// ---- DUTs/UR_6_T2O_IntRegisters/UR_6_T2O_IntRegisters.TcDUT
TYPE UR_6_T2O_IntRegisters :
STRUCT
INT0:ARRAY[0..3] OF BYTE;
INT1:ARRAY[0..3] OF BYTE;
INT2:ARRAY[0..3] OF BYTE;
INT3:ARRAY[0..3] OF BYTE;
INT4:ARRAY[0..3] OF BYTE;
INT5:ARRAY[0..3] OF BYTE;
INT6:ARRAY[0..3] OF BYTE;
INT7:ARRAY[0..3] OF BYTE;
INT8:ARRAY[0..3] OF BYTE;
INT9:ARRAY[0..3] OF BYTE;
INT10:ARRAY[0..3] OF BYTE;
INT11:ARRAY[0..3] OF BYTE;
INT12:ARRAY[0..3] OF BYTE;
INT13:ARRAY[0..3] OF BYTE;
INT14:ARRAY[0..3] OF BYTE;
INT15:ARRAY[0..3] OF BYTE;
INT16:ARRAY[0..3] OF BYTE;
INT17:ARRAY[0..3] OF BYTE;
INT18:ARRAY[0..3] OF BYTE;
INT19:ARRAY[0..3] OF BYTE;
INT20:ARRAY[0..3] OF BYTE;
INT21:ARRAY[0..3] OF BYTE;
INT22:ARRAY[0..3] OF BYTE;
INT23:ARRAY[0..3] OF BYTE;
END_STRUCT
END_TYPE

// ---- DUTs/UR_7_T2O_FloatRegisters/UR_7_T2O_FloatRegisters.TcDUT
TYPE UR_7_T2O_FloatRegisters :
	
STRUCT
FLOAT0:ARRAY[0..3] OF BYTE;
FLOAT1:ARRAY[0..3] OF BYTE;
FLOAT2:ARRAY[0..3] OF BYTE;
FLOAT3:ARRAY[0..3] OF BYTE;
FLOAT4:ARRAY[0..3] OF BYTE;
FLOAT5:ARRAY[0..3] OF BYTE;
FLOAT6:ARRAY[0..3] OF BYTE;
FLOAT7:ARRAY[0..3] OF BYTE;
FLOAT8:ARRAY[0..3] OF BYTE;
FLOAT9:ARRAY[0..3] OF BYTE;
FLOAT10:ARRAY[0..3] OF BYTE;
FLOAT11:ARRAY[0..3] OF BYTE;
FLOAT12:ARRAY[0..3] OF BYTE;
FLOAT13:ARRAY[0..3] OF BYTE;
FLOAT14:ARRAY[0..3] OF BYTE;
FLOAT15:ARRAY[0..3] OF BYTE;
FLOAT16:ARRAY[0..3] OF BYTE;
FLOAT17:ARRAY[0..3] OF BYTE;
FLOAT18:ARRAY[0..3] OF BYTE;
FLOAT19:ARRAY[0..3] OF BYTE;
FLOAT20:ARRAY[0..3] OF BYTE;
FLOAT21:ARRAY[0..3] OF BYTE;
FLOAT22:ARRAY[0..3] OF BYTE;
FLOAT23:ARRAY[0..3] OF BYTE;
END_STRUCT
END_TYPE

// ---- DUTs/UR_9_O2T_Registers/UR_9_O2T_Registers.TcDUT
TYPE UR_9_O2T_Registers :
STRUCT
	  Bits : UR_O2T_bits;
      Ints : UR_O2T_int;
      Floats : UR_O2T_floats;
END_STRUCT
END_TYPE

// ---- DUTs/UR_9_O2T_Registers/UR_O2T_bits.TcDUT
TYPE UR_O2T_bits :
   STRUCT
	B0:BIT;
	B1:BIT;
	B2:BIT;
	B3:BIT;
	B4:BIT;
	B5:BIT;
	B6:BIT;
	B7:BIT;
	B8:BIT;
	B9:BIT;
	B10:BIT;
	B11:BIT;
	B12:BIT;
	B13:BIT;
	B14:BIT;
	B15:BIT;
	B16:BIT;
	B17:BIT;
	B18:BIT;
	B19:BIT;
	B20:BIT;
	B21:BIT;
	B22:BIT;
	B23:BIT;
	B24:BIT;
	B25:BIT;
	B26:BIT;
	B27:BIT;
	B28:BIT;
	B29:BIT;
	B30:BIT;
	B31:BIT;
   END_STRUCT
END_TYPE

// ---- DUTs/UR_9_O2T_Registers/UR_O2T_floats.TcDUT
TYPE UR_O2T_floats :
STRUCT
FLOAT0:ARRAY[0..3] OF BYTE;
FLOAT1:ARRAY[0..3] OF BYTE;
FLOAT2:ARRAY[0..3] OF BYTE;
FLOAT3:ARRAY[0..3] OF BYTE;
FLOAT4:ARRAY[0..3] OF BYTE;
FLOAT5:ARRAY[0..3] OF BYTE;
FLOAT6:ARRAY[0..3] OF BYTE;
FLOAT7:ARRAY[0..3] OF BYTE;
FLOAT8:ARRAY[0..3] OF BYTE;
FLOAT9:ARRAY[0..3] OF BYTE;
FLOAT10:ARRAY[0..3] OF BYTE;
FLOAT11:ARRAY[0..3] OF BYTE;
END_STRUCT
END_TYPE

// ---- DUTs/UR_9_O2T_Registers/UR_O2T_int.TcDUT
TYPE UR_O2T_int :
STRUCT
INT0:ARRAY[0..3] OF BYTE;
INT1:ARRAY[0..3] OF BYTE;
INT2:ARRAY[0..3] OF BYTE;
INT3:ARRAY[0..3] OF BYTE;
INT4:ARRAY[0..3] OF BYTE;
INT5:ARRAY[0..3] OF BYTE;
INT6:ARRAY[0..3] OF BYTE;
INT7:ARRAY[0..3] OF BYTE;
INT8:ARRAY[0..3] OF BYTE;
INT9:ARRAY[0..3] OF BYTE;
INT10:ARRAY[0..3] OF BYTE;
INT11:ARRAY[0..3] OF BYTE;
END_STRUCT
END_TYPE

// ---- DUTs/Vision Struct/ck_real_flag_data.TcDUT
//struct to return values from POUS->Vision_functions->wr_real_value f
TYPE ck_real_flag_data :
STRUCT
	Flag : BOOL;
	Value : REAL;
END_STRUCT
END_TYPE

// ---- DUTs/Vision Struct/Vision_data.TcDUT
//struct to save vision real values system
TYPE Vision_data :
STRUCT
Val1 : REAL:= -1;
Val2 : REAL:= -1;
Val3 : REAL:= -1;
END_STRUCT
END_TYPE

// ---- DUTs/Vision Struct/Vision_flags.TcDUT
//struct to save vision flags values system
TYPE Vision_flags :
STRUCT
Flag1 :BOOL:=FALSE;	
Flag2 :BOOL:=FALSE;	
Flag3 :BOOL:=FALSE;	
END_STRUCT
END_TYPE

// ---- DUTs/Vision Struct/Vision_int_state.TcDUT
TYPE Vision_int_state :
STRUCT
	Val1 : INT:= -1;
	Val2 : INT:= -1;
	Val3 : INT:= -1;
END_STRUCT
END_TYPE

// ---- GVLs/MainProg Params/Constans/VFUNCTION.TcGVL
{attribute 'qualified_only'}
VAR_GLOBAL CONSTANT
	 	
	TEST:INT := 1; //test state one by one
	NORM:INT := 2; // normal functionality
	MOVEMENTS:INT := 3; // test just movements
	CK_COMUNICATIONS:INT := 4; // test all comunication
	POWEROFF:INT := 5; // prepare to poweroff the system
END_VAR

// ---- GVLs/MainProg Params/Constans/_FUNCTION.TcGVL
{attribute 'qualified_only'}
VAR_GLOBAL CONSTANT
	 	
	TEST:INT := 1; //test state one by one
	NORM:INT := 2; // normal functionality
	MOVEMENTS:INT := 3; // test just movements
	CK_COMUNICATIONS:INT := 4; // test all comunication
	POWEROFF:INT := 5; // prepare to poweroff the system
END_VAR

// ---- GVLs/MainProg Params/Variables/GLV_USER_FUN.TcGVL
{attribute 'qualified_only'}
VAR_GLOBAL RETAIN
		Value :INT:=2;
END_VAR

// ---- GVLs/miscellaneus/data_to_robot.TcGVL
{attribute 'qualified_only'}
VAR_GLOBAL
	head_roll_right : REAL;
	head_roll_left : REAL;
	
	
END_VAR

// ---- GVLs/miscellaneus/Global_actual_velocity.TcGVL
{attribute 'qualified_only'}
VAR_GLOBAL
	actual_velocity AT%I*: DINT;

	
	
	
END_VAR

// ---- GVLs/QRob/QrCts.TcGVL
{attribute 'qualified_only'}
VAR_GLOBAL CONSTANT
	MOVESTATE_INIT :INT:= 1;
	
	MOVESTATE_ENABLE :INT:= 2;
	MOVESTATE_ENABLE_F :INT:= 21;
	
	MOVESTATE_ERROR :INT:=3;
	MOVESTATE_ERROR_F :INT:=31;
	
	MOVESTATE_RESET : INT:=4;
	MOVESTATE_RESET_F : INT:=41;
	
	MOVESTATE_MOVABS : INT:=5;
	MOVESTATE_MOVABS_I :INT:=50;
	MOVESTATE_MOVABS_F :INT:=51;
	
	MOVESTATE_HOME:  INT:=6;
	MOVESTATE_HOME_I:  INT:=60;
	MOVESTATE_HOME_F:  INT:=61;
	
	MOVESTATE_CTR_W : INT := 7;
	MOVESTATE_CTR_W_I : INT := 70;
	MOVESTATE_CTR_W_F : INT := 71;
	
	MOVESTATE_TORQUE : INT := 8;
	MOVESTATE_TORQUE_I : INT := 80;
	MOVESTATE_TORQUE_F : INT := 81;
	
	
	MOVESTATE_RELIEF : INT := 9;
	MOVESTATE_RELIEF_I : INT := 90;
	MOVESTATE_RELIEF_F : INT := 91;
	
	OFFSETHOME : INT := 15;
	OFFSETHOME_I : INT := 150;
	OFFSETHOME_F : INT := 151;
	
END_VAR

// ---- GVLs/QRob/Variables/Global_Servo.TcGVL
{attribute 'qualified_only'}
VAR_GLOBAL
	Axis1 : AXIS_REF;
	
END_VAR

// ---- GVLs/QRob/Variables/QrRetVarState.TcGVL
{attribute 'qualified_only'}
VAR_GLOBAL RETAIN
	Actual_GLV_State :INT:=-1;
	Actual_In_State: INT:=-1;
	Actual_POs :REAL:=0;
END_VAR

// ---- GVLs/Robot Params/Constans/RCts.TcGVL
{attribute 'qualified_only'}
VAR_GLOBAL CONSTANT


// 


   

//############### CS.UR3 CONSTANTS STATES ###################
//########################################################
	RESET_STATE:INT:=-1;
	//CS.UR3 states
	UR3:INT:=3;
	UR3Home:INT := 30;
	UR3Home_I :INT:= 300;
	UR3Home_F :INT:= 301;
	
    UR3CatchSeparator:INT := 31;
	UR3CatchSeparator_I:INT := 310;
	UR3CatchSeparator_F:INT := 311;
	
	UR3Move:INT := 32;
	UR3Move_I:INT := 320;	
	UR3Move_F:INT := 321;
	
	UR3DropBench:INT := 33;
	UR3DropBench_I:INT := 330;
	UR3DropBench_F:INT := 331;
	
	
	UR3Correct_Insertion :INT:=39;
	UR3Correct_Insertion_I :INT:=390;
	UR3Correct_Insertion_F :INT:=391;
	
	UR3RotateSeparator:INT := 34;
	UR3RotateSeparator_I:INT := 340;
	UR3RotateSeparator_F:INT := 341;
	
	UR3RotateDropCable:INT := 35;
	UR3RotateDropCable_I:INT := 350;
	UR3RotateDropCable_F:INT := 351;
	
	UR3DropCable:INT := 36;
	UR3DropCable_I:INT := 360;
	UR3DropCable_F:INT := 361;
	
	UR3Return:INT := 37;
	UR3Return_I:INT := 370;
	UR3Return_F:INT := 371;
	
//############### CS.UR5 CONSTANTS STATES ###################
//########################################################
 

    UR_DATA_SEND : INT :=-2;
	
	UR5:INT:=5;
	
	UR5Home:INT := 50;
	UR5Home_I :INT:= 500;
	UR5Home_F :INT:= 501;
	
    UR5Camera1:INT := 51;
	UR5Camera1_I:INT := 510;
	UR5Camera1_F:INT := 511;
	
	UR5DropHead:INT := 52;
	UR5DropHead_I:INT := 520;	
	UR5DropHead_F:INT := 521;
	
	UR5Camera2:INT := 53;
	UR5Camera2_I:INT := 530;
	UR5Camera2_F:INT := 531;
	
	UR5UpCamera1:INT := 54;
	UR5UpCamera1_I:INT := 540;
	UR5UpCamera1_F:INT := 541;
	
	UR5TakeBuffer:INT := 55;
	UR5TakeBuffer_I:INT := 550;
	UR5TakeBuffer_F:INT := 551;
	
	UR5UpCamera2:INT := 56;
	UR5UpCamera2_I:INT := 560;
	UR5UpCamera2_F:INT := 561;
	
	UR5Return:INT := 57;
	UR5Return_I:INT := 570;
	UR5Return_F:INT := 571;

	/// to ck new values
	UR5CkPosSepator : INT := 69;
	UR5CkPosSepator_I: INT := 690;
	UR5CkPosSepator_F: INT := 691;
	
	UR5CtrHeadTurnR : INT := 70;
	UR5CtrHeadTurnR_I : INT := 700;
	UR5CtrHeadTurnR_F : INT := 701;
	
	
	UR5CtrHeadTurnL : INT := 71;
	UR5CtrHeadTurnL_I : INT := 710;
	UR5CtrHeadTurnL_F : INT := 711;
	
	
	UR5CtrCamPos1:INT:=58;
	UR5CtrCamPos2:INT:=60;
	UR5CtrCamPos3:INT:=62;
	UR5CtrCamPos4:INT:=64;
	UR5CtrCamPos:INT:=582;
	UR5CtrCamPos_I:INT:=580;
	UR5CtrCamPos_F:INT:=581;

	UR5MoveToNut:INT:=592;	
	UR5MoveToNut_I:INT:=590;
	UR5MoveToNut_F:INT:=591;
	UR5MoveToNut1:INT:=59;
	UR5MoveToNut2:INT:=61;
	UR5MoveToNut3:INT:=63;
	UR5MoveToNut4:INT:=65;
	
	UR5Correct_Insertion :INT:=73;
	UR5Correct_Insertion_I :INT:=730;
	UR5Correct_Insertion_F :INT:=731;

	
	UR5UnScrew:INT:=66;
	UR5UnScrew_I:INT:=5100;
	UR5UnScrew_F:INT:=5101;
	
	
	UR5ScrewHigh:INT:=72;
	UR5ScrewHigh_I:INT:=5130;
	UR5ScrewHigh_F:INT:=5131;
	
	UR5Screw:INT:=67;
	UR5Screw_I:INT:=5110;
	UR5Screw_F:INT:=5111;
	
	UR5UpRobotAs:INT:=68;
	UR5UpRobotAs_I:INT:=5120;
	UR5UpRobotAs_F:INT:=5121;
	

END_VAR

// ---- GVLs/Robot Params/Variables/Robot_UR5.TcGVL
{attribute 'qualified_only'}
VAR_GLOBAL
//variables para enviar al robot
UR_inputs AT%Q* : UR_9_O2T_Registers;
UR_inputs_2 AT%Q* : UR_10_O2T_Registers;

//variables para recibir del robot
UR_outputs AT%I*:UR_5_T2O_BitRegisters;
UR_outputs_int AT%I*:UR_6_T2O_IntRegisters;
UR_outputs_float AT%I*:UR_7_T2O_FloatRegisters;

UR_TCP AT%I*:UR_4_T2O_TCP;

UR_JOINS AT%I*:UR_3_T2O_Joints;


END_VAR 

////variables para enviar al robot
//UR_inputs AT%Q* : UR_9_O2T_Registers;
//UR_inputs_2 AT%Q* : UR_10_O2T_Registers;
////variables para recibir del robot
//UR_outputs AT%I*:UR_5_T2O_BitRegisters;
//UR_outputs_int AT%I*:UR_6_T2O_IntRegisters;

//UR_TCP AT%I*:UR_4_T2O_TCP;

//UR_JOINS AT%I*:UR_3_T2O_Joints;

//UR_float_out AT%I*:UR_7_T2O;

// ---- GVLs/Robot Params/Variables/Robot_UR3.TcGVL
{attribute 'qualified_only'}
VAR_GLOBAL
	
//variables para enviar al robot
UR_inputs AT%Q* : UR_9_O2T_Registers;


//variables para recibir del robot
UR_outputs AT%I*:UR_5_T2O_BitRegisters;
UR_outputs_int AT%I*:UR_6_T2O_IntRegisters;
UR_outputs_float AT%I*:UR_7_T2O_FloatRegisters;

UR_TCP AT%I*:UR_4_T2O_TCP;
UR_JOINS AT%I*:UR_3_T2O_Joints;


	UR_float_out: INT;
END_VAR

// ---- GVLs/Robot Params/Variables/UR3RetVarState.TcGVL
{attribute 'qualified_only'}
VAR_GLOBAL RETAIN
	Actual_GLV_State :INT:=-1;
	Actual_In_State: INT:=-1;
END_VAR

// ---- GVLs/Vision Params/Constants/VCts.TcGVL
{attribute 'qualified_only'}
VAR_GLOBAL CONSTANT
	
	//constans to exec respective function into vision system
	
	RESET : INT :=-1;
	CX_VALUE:INT:=1;
	CY_VALUE:INT:=2;
	NUT_VALUE:INT:=3;
	HEAD_RIGTH_VALUE : INT:= 4;
	HEAD_LEFT_VALUE : INT:= 5;
	SEP_POS_VALUE: INT:= 6;
	
	//separator variables 
	Separador_correct:INT:=7;
	Separador_turned:INT:=8;
	
	//constans to state machine
	SeparatorPos:INT := 10;
	SeparatorPos_I:INT := 100;
	SeparatorPos_F:INT := 101;
	
	SeparatorRot_R:INT:= 11;
	SeparatorRot_R_I:INT:= 110;
	SeparatorRot_R_F:INT:= 111;
	
	SeparatorRot_L:INT:= 12;
	SeparatorRot_L_I:INT:= 120;
	SeparatorRot_L_F:INT:= 121;
	
	SeparatorNut:INT:=13;
	SeparatorNut_I:INT:=130;
	SeparatorNut_F:INT:=131;
	
	SeparatorHole:INT:=14;
	SeparatorHole_I:INT:=140;
	SeparatorHole_F:INT:=141;
	
	
END_VAR

// ---- GVLs/Vision Params/Structs/Vision_struct.TcGVL
{attribute 'qualified_only'}
VAR_GLOBAL

//variables to start head rigth roll vision process (PLC->vision)
//Get_img_head_rigth_rot : Vision_flags;
//variables to start head left roll vision process (PLC->vision)
//Get_img_head_left_rot : Vision_flags;
//variables to start nut vision process (PLC->vision)
//Get_img_nut :Vision_flags;	
//variables to start orifice vision process (PLC->vision)
//Get_img_orifice :Vision_flags;	
//variables to start check separator position
//Get_img_sep_pos :Vision_flags;	

//variables to read global and internal state from vision system
States_out : Vision_int_state;
States_in : Vision_int_state;

//variables to ck  vision process (vision->PLC)  
//Ck_finish_procees :Vision_flags;
// variables to get position of separator from vision system
Pos_sep : Vision_data;
// variables to get cx value from vision system
Cx_value_nut : Vision_data;
// variables to get cy value from vision system
Cy_value_nut : Vision_data;
// variables to get cx value from vision system
Cx_value_hole : Vision_data;
// variables to get cy value from vision system
Cy_value_hole : Vision_data;
// variables to get turn_nut value from vision system
Nut_turn_value :Vision_data;
// variables to get head_rigth value from vision system
Head_rigth_value	:Vision_data;
// variables to get head_left value from vision system
Head_left_value	:Vision_data;
	Get_img_sep_pos: INT;
END_VAR

// ---- GVLs/Vision Params/Variables/VisionRetVarState.TcGVL
{attribute 'qualified_only'}
VAR_GLOBAL RETAIN
	Actual_GLV_State :INT:=-1;
	Actual_In_State: INT:=-1;
END_VAR

// ---- POUs/POUs/MASTER_CTR.TcPOU
PROGRAM MASTER_CTR
VAR
	//check status from finish state

	finish_state : BOOL:=FALSE;
	//var state to norm mode
	STATE :INT:=-1;
    //
	home_ur3 : BOOL ;
	home_ur5 : BOOL ;
	//instance of Qrob
	//QRob_StateMachine : QRob_StateMachine;
	

	
	

	//var to ck pictures of separator position
	Pos_Ck_Finish : BOOL ;
	sep_pos_data : ck_real_flag_data;
	Neural_Net_val : ARRAY[0..5] OF REAL;
	aux_for : INT;

	
	
	//vars to get the rigt/left rotation 
	sep_rot_rigth_data :ck_real_flag_data;	
	sep_rot_left_data :ck_real_flag_data;
	
	
	//var to check the error cam optical center and robot position
	cx_vision_data : ck_real_flag_data;
	cy_vision_data : ck_real_flag_data;
	nut_turn_data : ck_real_flag_data;
	Cam_center_ok : BOOL := FALSE;
	error_vision : REAL := 1;

	//var to qrob 
	turn_aux_int : INT := 0;
	turn_aux_float : REAL:= 0;
	Pos_qrob_buffer :REAL;	
	Torque_SetPoint: INT;
	

	//var to ck screw finish
	screw_finish : BOOL ;
	
	//var to ck return robots
	return_ur5 : BOOL;
	return_ur3 : BOOL;
	
	//var to qrob_home;
	qrob_home_flag : BOOL;
	

	
	//var to ck correct operation tool into nut 
	ck_operation : BOOL ;
	
	//data betweem robots 
	UR3_norm_force : REAL;
    UR5_norm_force : REAL;
	
	ELIF: INT;
	MoveAbsAxis1: INT;
	sleep7: INT;
	t: INT;
	
	
			//var to control the global state
	Global_State : INT := -1;
		//var to select cam pos 
	cam_pos : INT := -1;
	sleepS8: INT;
END_VAR

VAR_INPUT
	//vars to control the main stata machine
	  user_select_state : INT:=-1;
	  user_init: BOOL:=FALSE;
      User_Test_Sate :INT:=-1;
	  EMERGENCY_STOP :BOOL:=FALSE;
	  
END_VAR

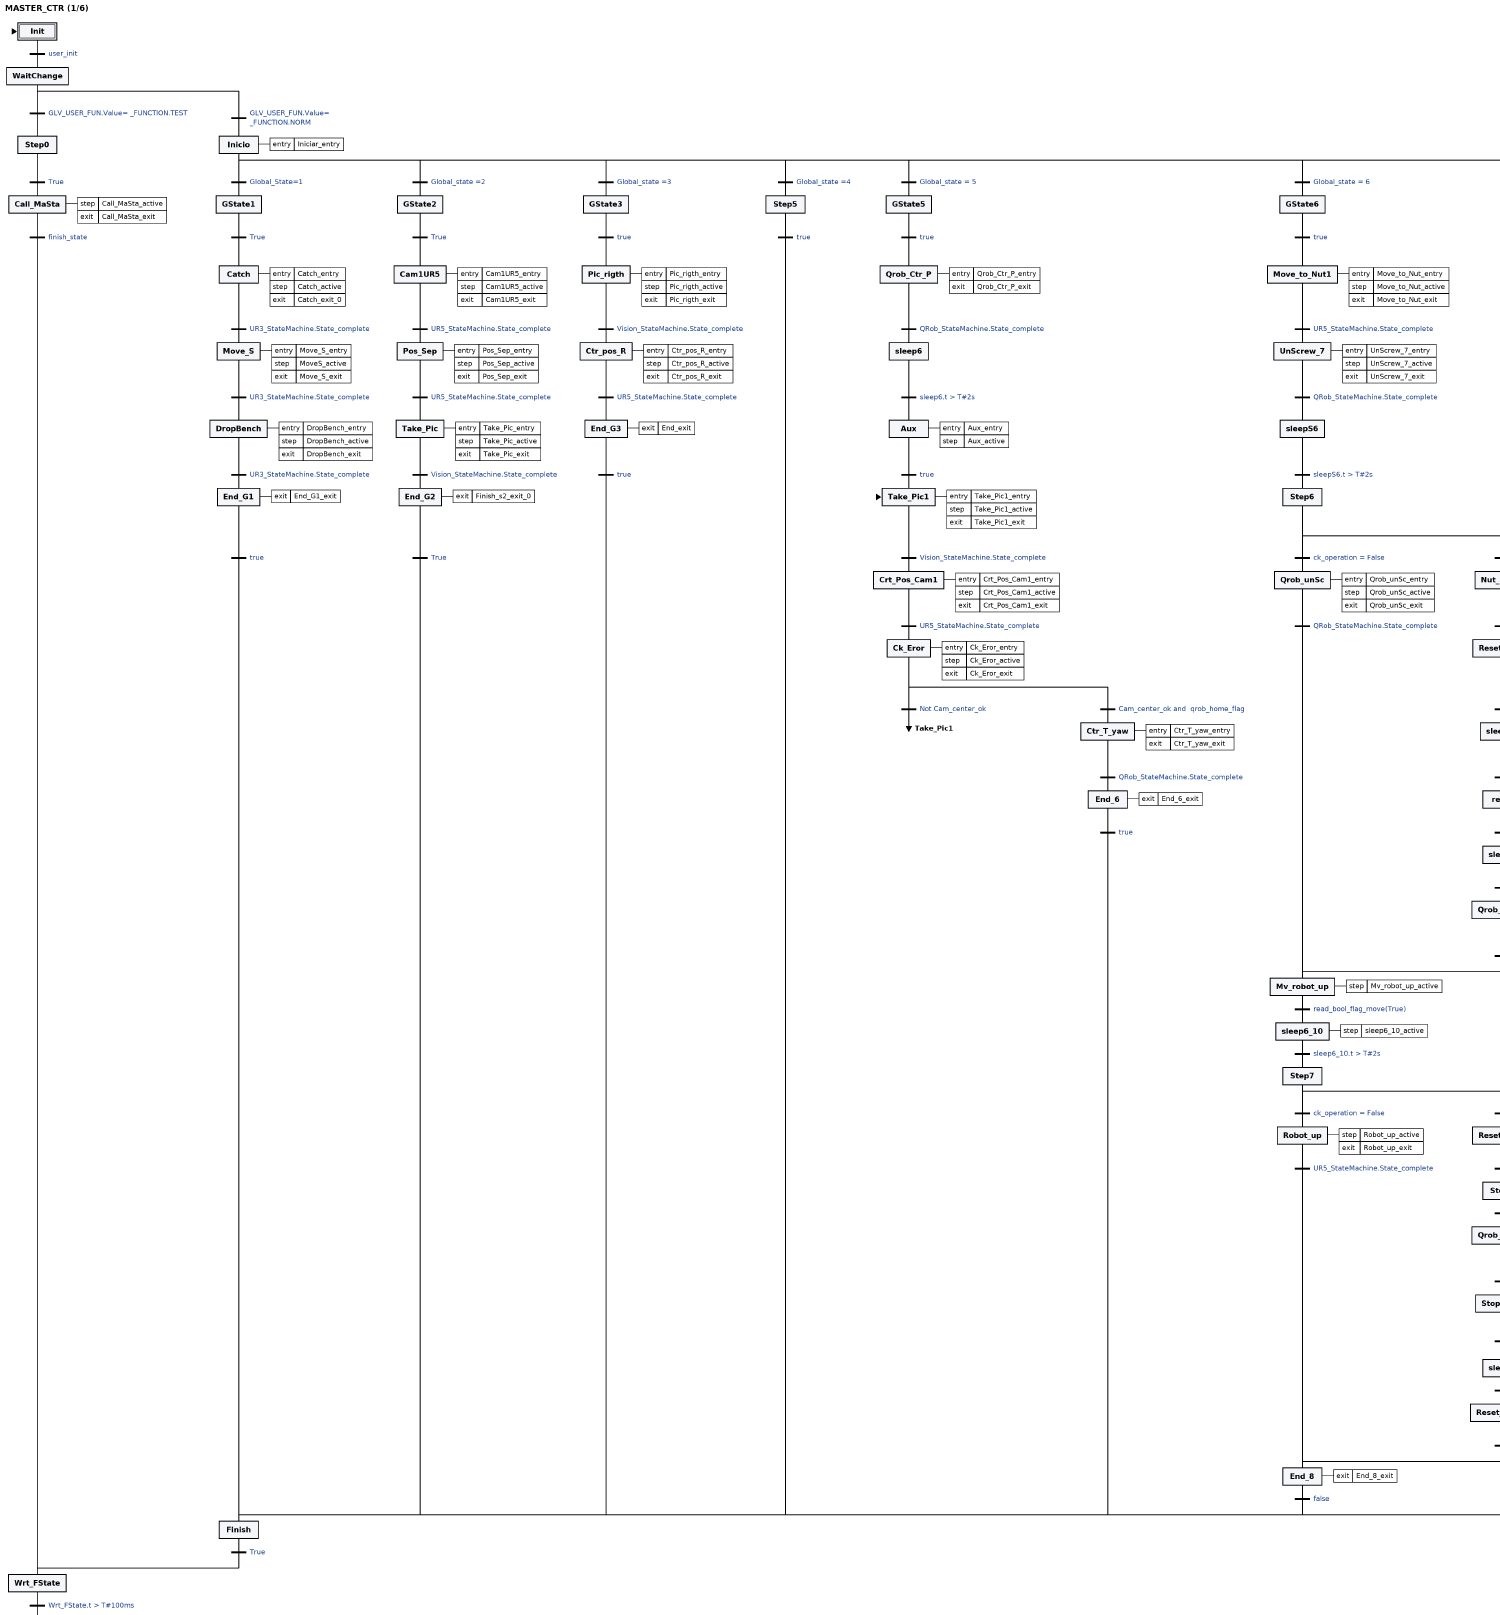
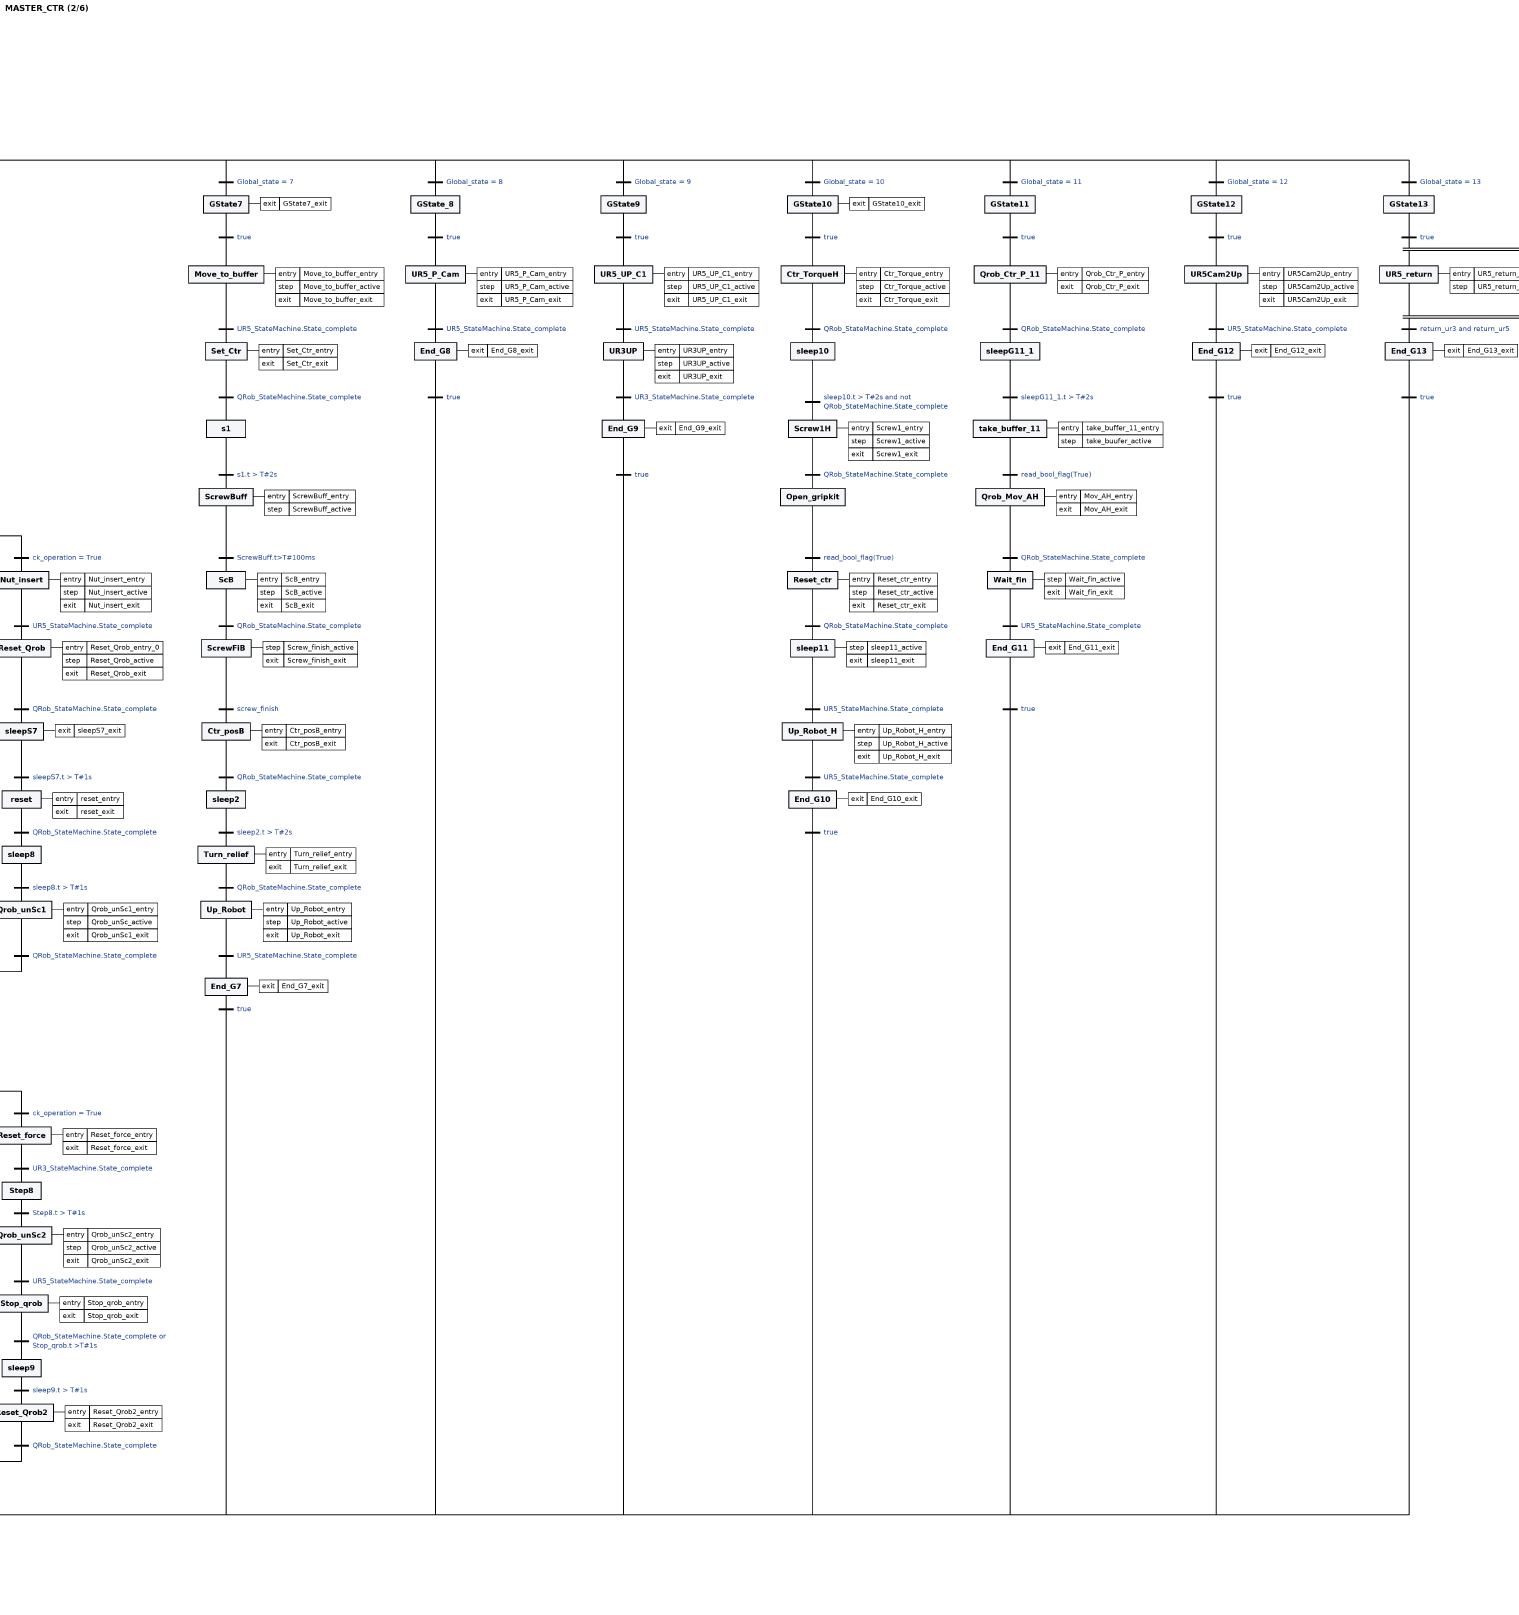
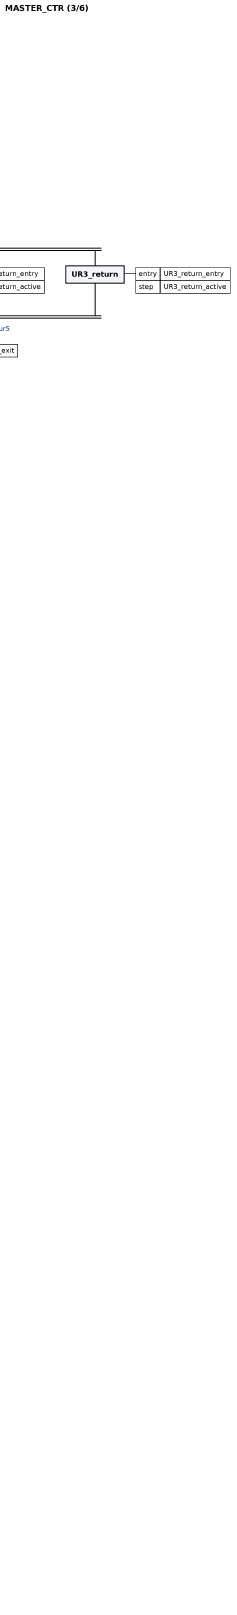
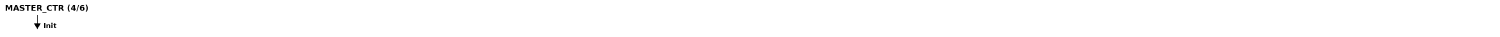
INITIAL_STEP Init:
END_STEP
TRANSITION FROM Init TO WaitChange
    := user_init;
END_TRANSITION
STEP WaitChange:
END_STEP
TRANSITION FROM WaitChange TO Step0
    := GLV_USER_FUN.Value= _FUNCTION.TEST;
END_TRANSITION
// macro TestMode begins
STEP Step0:
END_STEP
TRANSITION FROM Step0 TO Call_MaSta
    := True;
END_TRANSITION
STEP Call_MaSta:
    Call_MaSta_active(N);  // step action
    Call_MaSta_exit(P0);  // exit action
END_STEP
TRANSITION FROM Call_MaSta TO Wrt_FState
    := finish_state;
END_TRANSITION
TRANSITION FROM WaitChange TO Inicio
    := GLV_USER_FUN.Value= _FUNCTION.NORM;
END_TRANSITION
// macro NormMode begins
STEP Inicio:
    Iniciar_entry(P1);  // entry action
END_STEP
TRANSITION FROM Inicio TO GState1
    := Global_State=1;
END_TRANSITION
// macro MovSeparator begins
STEP GState1:
END_STEP
TRANSITION FROM GState1 TO Catch
    := True;
END_TRANSITION
STEP Catch:
    Catch_entry(P1);  // entry action
    Catch_active(N);  // step action
    Catch_exit_0(P0);  // exit action
END_STEP
TRANSITION FROM Catch TO Move_S
    := UR3_StateMachine.State_complete;
END_TRANSITION
STEP Move_S:
    Move_S_entry(P1);  // entry action
    MoveS_active(N);  // step action
    Move_S_exit(P0);  // exit action
END_STEP
TRANSITION FROM Move_S TO DropBench
    := UR3_StateMachine.State_complete;
END_TRANSITION
STEP DropBench:
    DropBench_entry(P1);  // entry action
    DropBench_active(N);  // step action
    DropBench_exit(P0);  // exit action
END_STEP
TRANSITION FROM DropBench TO End_G1
    := UR3_StateMachine.State_complete;
END_TRANSITION
STEP End_G1:
    End_G1_exit(P0);  // exit action
END_STEP
TRANSITION FROM End_G1 TO Finish
    := true;
END_TRANSITION
TRANSITION FROM Inicio TO GState2
    := Global_state =2;
END_TRANSITION
// macro CkPos begins
STEP GState2:
END_STEP
TRANSITION FROM GState2 TO Cam1UR5
    := True;
END_TRANSITION
STEP Cam1UR5:
    Cam1UR5_entry(P1);  // entry action
    Cam1UR5_active(N);  // step action
    Cam1UR5_exit(P0);  // exit action
END_STEP
TRANSITION FROM Cam1UR5 TO Pos_Sep
    := UR5_StateMachine.State_complete;
END_TRANSITION
STEP Pos_Sep:
    Pos_Sep_entry(P1);  // entry action
    Pos_Sep_active(N);  // step action
    Pos_Sep_exit(P0);  // exit action
END_STEP
TRANSITION FROM Pos_Sep TO Take_Pic
    := UR5_StateMachine.State_complete;
END_TRANSITION
STEP Take_Pic:
    Take_Pic_entry(P1);  // entry action
    Take_Pic_active(N);  // step action
    Take_Pic_exit(P0);  // exit action
END_STEP
TRANSITION FROM Take_Pic TO End_G2
    := Vision_StateMachine.State_complete;
END_TRANSITION
STEP End_G2:
    Finish_s2_exit_0(P0);  // exit action
END_STEP
TRANSITION FROM End_G2 TO Finish
    := True;
END_TRANSITION
TRANSITION FROM Inicio TO GState3
    := Global_state =3;
END_TRANSITION
// macro Ctr_Head_rot begins
STEP GState3:
END_STEP
TRANSITION FROM GState3 TO Pic_rigth
    := true;
END_TRANSITION
STEP Pic_rigth:
    Pic_rigth_entry(P1);  // entry action
    Pic_rigth_active(N);  // step action
    Pic_rigth_exit(P0);  // exit action
END_STEP
TRANSITION FROM Pic_rigth TO Ctr_pos_R
    := Vision_StateMachine.State_complete;
END_TRANSITION
STEP Ctr_pos_R:
    Ctr_pos_R_entry(P1);  // entry action
    Ctr_pos_R_active(N);  // step action
    Ctr_pos_R_exit(P0);  // exit action
END_STEP
TRANSITION FROM Ctr_pos_R TO End_G3
    := UR5_StateMachine.State_complete;
END_TRANSITION
STEP End_G3:
    End_exit(P0);  // exit action
END_STEP
TRANSITION FROM End_G3 TO Finish
    := true;
END_TRANSITION
TRANSITION FROM Inicio TO Step5
    := Global_state =4;
END_TRANSITION
// macro Rot_Sepa begins
STEP Step5:
END_STEP
TRANSITION FROM Step5 TO Finish
    := true;
END_TRANSITION
TRANSITION FROM Inicio TO GState5
    := Global_state = 5;
END_TRANSITION
// macro Ctr_CaM begins
STEP GState5:
END_STEP
TRANSITION FROM GState5 TO Qrob_Ctr_P
    := true;
END_TRANSITION
STEP Qrob_Ctr_P:
    Qrob_Ctr_P_entry(P1);  // entry action
    Qrob_Ctr_P_exit(P0);  // exit action
END_STEP
TRANSITION FROM Qrob_Ctr_P TO sleep6
    := QRob_StateMachine.State_complete;
END_TRANSITION
STEP sleep6:
END_STEP
TRANSITION FROM sleep6 TO Aux
    := sleep6.t > T#2s;
END_TRANSITION
STEP Aux:
    Aux_entry(P1);  // entry action
    Aux_active(N);  // step action
END_STEP
TRANSITION FROM Aux TO Take_Pic1
    := true;
END_TRANSITION
STEP Take_Pic1:
    Take_Pic1_entry(P1);  // entry action
    Take_Pic1_active(N);  // step action
    Take_Pic1_exit(P0);  // exit action
END_STEP
TRANSITION FROM Take_Pic1 TO Crt_Pos_Cam1
    := Vision_StateMachine.State_complete;
END_TRANSITION
STEP Crt_Pos_Cam1:
    Crt_Pos_Cam1_entry(P1);  // entry action
    Crt_Pos_Cam1_active(N);  // step action
    Crt_Pos_Cam1_exit(P0);  // exit action
END_STEP
TRANSITION FROM Crt_Pos_Cam1 TO Ck_Eror
    := UR5_StateMachine.State_complete;
END_TRANSITION
STEP Ck_Eror:
    Ck_Eror_entry(P1);  // entry action
    Ck_Eror_active(N);  // step action
    Ck_Eror_exit(P0);  // exit action
END_STEP
TRANSITION FROM Ck_Eror TO Take_Pic1
    := Not Cam_center_ok;
END_TRANSITION
TRANSITION FROM Ck_Eror TO Ctr_T_yaw
    := Cam_center_ok and qrob_home_flag;
END_TRANSITION
STEP Ctr_T_yaw:
    Ctr_T_yaw_entry(P1);  // entry action
    Ctr_T_yaw_exit(P0);  // exit action
END_STEP
TRANSITION FROM Ctr_T_yaw TO End_6
    := QRob_StateMachine.State_complete;
END_TRANSITION
STEP End_6:
    End_6_exit(P0);  // exit action
END_STEP
TRANSITION FROM End_6 TO Finish
    := true;
END_TRANSITION
TRANSITION FROM Inicio TO GState6
    := Global_state = 6;
END_TRANSITION
// macro UnScrew begins
STEP GState6:
END_STEP
TRANSITION FROM GState6 TO Move_to_Nut1
    := true;
END_TRANSITION
STEP Move_to_Nut1:
    Move_to_Nut_entry(P1);  // entry action
    Move_to_Nut_active(N);  // step action
    Move_to_Nut_exit(P0);  // exit action
END_STEP
TRANSITION FROM Move_to_Nut1 TO UnScrew_7
    := UR5_StateMachine.State_complete;
END_TRANSITION
STEP UnScrew_7:
    UnScrew_7_entry(P1);  // entry action
    UnScrew_7_active(N);  // step action
    UnScrew_7_exit(P0);  // exit action
END_STEP
TRANSITION FROM UnScrew_7 TO sleepS6
    := QRob_StateMachine.State_complete;
END_TRANSITION
STEP sleepS6:
END_STEP
TRANSITION FROM sleepS6 TO Step6
    := sleepS6.t > T#2s;
END_TRANSITION
STEP Step6:
END_STEP
TRANSITION FROM Step6 TO Qrob_unSc
    := ck_operation = False;
END_TRANSITION
STEP Qrob_unSc:
    Qrob_unSc_entry(P1);  // entry action
    Qrob_unSc_active(N);  // step action
    Qrob_unSc_exit(P0);  // exit action
END_STEP
TRANSITION FROM Qrob_unSc TO Mv_robot_up
    := QRob_StateMachine.State_complete;
END_TRANSITION
TRANSITION FROM Step6 TO Nut_insert
    := ck_operation = True;
END_TRANSITION
STEP Nut_insert:
    Nut_insert_entry(P1);  // entry action
    Nut_insert_active(N);  // step action
    Nut_insert_exit(P0);  // exit action
END_STEP
TRANSITION FROM Nut_insert TO Reset_Qrob
    := UR5_StateMachine.State_complete;
END_TRANSITION
STEP Reset_Qrob:
    Reset_Qrob_entry_0(P1);  // entry action
    Reset_Qrob_active(N);  // step action
    Reset_Qrob_exit(P0);  // exit action
END_STEP
TRANSITION FROM Reset_Qrob TO sleepS7
    := QRob_StateMachine.State_complete;
END_TRANSITION
STEP sleepS7:
    sleepS7_exit(P0);  // exit action
END_STEP
TRANSITION FROM sleepS7 TO reset
    := sleepS7.t > T#1s;
END_TRANSITION
STEP reset:
    reset_entry(P1);  // entry action
    reset_exit(P0);  // exit action
END_STEP
TRANSITION FROM reset TO sleep8
    := QRob_StateMachine.State_complete;
END_TRANSITION
STEP sleep8:
END_STEP
TRANSITION FROM sleep8 TO Qrob_unSc1
    := sleep8.t > T#1s;
END_TRANSITION
STEP Qrob_unSc1:
    Qrob_unSc1_entry(P1);  // entry action
    Qrob_unSc_active(N);  // step action
    Qrob_unSc1_exit(P0);  // exit action
END_STEP
TRANSITION FROM Qrob_unSc1 TO Mv_robot_up
    := QRob_StateMachine.State_complete;
END_TRANSITION
STEP Mv_robot_up:
    Mv_robot_up_active(N);  // step action
END_STEP
TRANSITION FROM Mv_robot_up TO sleep6_10
    := read_bool_flag_move(True);
END_TRANSITION
STEP sleep6_10:
    sleep6_10_active(N);  // step action
END_STEP
TRANSITION FROM sleep6_10 TO Step7
    := sleep6_10.t > T#2s;
END_TRANSITION
STEP Step7:
END_STEP
TRANSITION FROM Step7 TO Robot_up
    := ck_operation = False;
END_TRANSITION
STEP Robot_up:
    Robot_up_active(N);  // step action
    Robot_up_exit(P0);  // exit action
END_STEP
TRANSITION FROM Robot_up TO End_8
    := UR5_StateMachine.State_complete;
END_TRANSITION
TRANSITION FROM Step7 TO Reset_force
    := ck_operation = True;
END_TRANSITION
STEP Reset_force:
    Reset_force_entry(P1);  // entry action
    Reset_force_exit(P0);  // exit action
END_STEP
TRANSITION FROM Reset_force TO Step8
    := UR3_StateMachine.State_complete;
END_TRANSITION
STEP Step8:
END_STEP
TRANSITION FROM Step8 TO Qrob_unSc2
    := Step8.t > T#1s;
END_TRANSITION
STEP Qrob_unSc2:
    Qrob_unSc2_entry(P1);  // entry action
    Qrob_unSc2_active(N);  // step action
    Qrob_unSc2_exit(P0);  // exit action
END_STEP
TRANSITION FROM Qrob_unSc2 TO Stop_qrob
    := UR5_StateMachine.State_complete;
END_TRANSITION
STEP Stop_qrob:
    Stop_qrob_entry(P1);  // entry action
    Stop_qrob_exit(P0);  // exit action
END_STEP
TRANSITION FROM Stop_qrob TO sleep9
    := QRob_StateMachine.State_complete or Stop_qrob.t >T#1s;
END_TRANSITION
STEP sleep9:
END_STEP
TRANSITION FROM sleep9 TO Reset_Qrob2
    := sleep9.t > T#1s;
END_TRANSITION
STEP Reset_Qrob2:
    Reset_Qrob2_entry(P1);  // entry action
    Reset_Qrob2_exit(P0);  // exit action
END_STEP
TRANSITION FROM Reset_Qrob2 TO End_8
    := QRob_StateMachine.State_complete;
END_TRANSITION
STEP End_8:
    End_8_exit(P0);  // exit action
END_STEP
TRANSITION FROM End_8 TO Finish
    := false;
END_TRANSITION
TRANSITION FROM Inicio TO GState7
    := Global_state = 7;
END_TRANSITION
// macro Buffer begins
STEP GState7:
    GState7_exit(P0);  // exit action
END_STEP
TRANSITION FROM GState7 TO Move_to_buffer
    := true;
END_TRANSITION
STEP Move_to_buffer:
    Move_to_buffer_entry(P1);  // entry action
    Move_to_buffer_active(N);  // step action
    Move_to_buffer_exit(P0);  // exit action
END_STEP
TRANSITION FROM Move_to_buffer TO Set_Ctr
    := UR5_StateMachine.State_complete;
END_TRANSITION
STEP Set_Ctr:
    Set_Ctr_entry(P1);  // entry action
    Set_Ctr_exit(P0);  // exit action
END_STEP
TRANSITION FROM Set_Ctr TO s1
    := QRob_StateMachine.State_complete;
END_TRANSITION
STEP s1:
END_STEP
TRANSITION FROM s1 TO ScrewBuff
    := s1.t > T#2s;
END_TRANSITION
STEP ScrewBuff:
    ScrewBuff_entry(P1);  // entry action
    ScrewBuff_active(N);  // step action
END_STEP
TRANSITION FROM ScrewBuff TO ScB
    := ScrewBuff.t>T#100ms;
END_TRANSITION
STEP ScB:
    ScB_entry(P1);  // entry action
    ScB_active(N);  // step action
    ScB_exit(P0);  // exit action
END_STEP
TRANSITION FROM ScB TO ScrewFiB
    := QRob_StateMachine.State_complete;
END_TRANSITION
STEP ScrewFiB:
    Screw_finish_active(N);  // step action
    Screw_finish_exit(P0);  // exit action
END_STEP
TRANSITION FROM ScrewFiB TO Ctr_posB
    := screw_finish;
END_TRANSITION
STEP Ctr_posB:
    Ctr_posB_entry(P1);  // entry action
    Ctr_posB_exit(P0);  // exit action
END_STEP
TRANSITION FROM Ctr_posB TO sleep2
    := QRob_StateMachine.State_complete;
END_TRANSITION
STEP sleep2:
END_STEP
TRANSITION FROM sleep2 TO Turn_relief
    := sleep2.t > T#2s;
END_TRANSITION
STEP Turn_relief:
    Turn_relief_entry(P1);  // entry action
    Turn_relief_exit(P0);  // exit action
END_STEP
TRANSITION FROM Turn_relief TO Up_Robot
    := QRob_StateMachine.State_complete;
END_TRANSITION
STEP Up_Robot:
    Up_Robot_entry(P1);  // entry action
    Up_Robot_active(N);  // step action
    Up_Robot_exit(P0);  // exit action
END_STEP
TRANSITION FROM Up_Robot TO End_G7
    := UR5_StateMachine.State_complete;
END_TRANSITION
STEP End_G7:
    End_G7_exit(P0);  // exit action
END_STEP
TRANSITION FROM End_G7 TO Finish
    := true;
END_TRANSITION
TRANSITION FROM Inicio TO GState_8
    := Global_state = 8;
END_TRANSITION
// macro CAM2 begins
STEP GState_8:
END_STEP
TRANSITION FROM GState_8 TO UR5_P_Cam
    := true;
END_TRANSITION
STEP UR5_P_Cam:
    UR5_P_Cam_entry(P1);  // entry action
    UR5_P_Cam_active(N);  // step action
    UR5_P_Cam_exit(P0);  // exit action
END_STEP
TRANSITION FROM UR5_P_Cam TO End_G8
    := UR5_StateMachine.State_complete;
END_TRANSITION
STEP End_G8:
    End_G8_exit(P0);  // exit action
END_STEP
TRANSITION FROM End_G8 TO Finish
    := true;
END_TRANSITION
TRANSITION FROM Inicio TO GState9
    := Global_state = 9;
END_TRANSITION
// macro Cam1Up begins
STEP GState9:
END_STEP
TRANSITION FROM GState9 TO UR5_UP_C1
    := true;
END_TRANSITION
STEP UR5_UP_C1:
    UR5_UP_C1_entry(P1);  // entry action
    UR5_UP_C1_active(N);  // step action
    UR5_UP_C1_exit(P0);  // exit action
END_STEP
TRANSITION FROM UR5_UP_C1 TO UR3UP
    := UR5_StateMachine.State_complete;
END_TRANSITION
STEP UR3UP:
    UR3UP_entry(P1);  // entry action
    UR3UP_active(N);  // step action
    UR3UP_exit(P0);  // exit action
END_STEP
TRANSITION FROM UR3UP TO End_G9
    := UR3_StateMachine.State_complete;
END_TRANSITION
STEP End_G9:
    End_G9_exit(P0);  // exit action
END_STEP
TRANSITION FROM End_G9 TO Finish
    := true;
END_TRANSITION
TRANSITION FROM Inicio TO GState10
    := Global_state = 10;
END_TRANSITION
// macro HighScrew begins
STEP GState10:
    GState10_exit(P0);  // exit action
END_STEP
TRANSITION FROM GState10 TO Ctr_TorqueH
    := true;
END_TRANSITION
STEP Ctr_TorqueH:
    Ctr_Torque_entry(P1);  // entry action
    Ctr_Torque_active(N);  // step action
    Ctr_Torque_exit(P0);  // exit action
END_STEP
TRANSITION FROM Ctr_TorqueH TO sleep10
    := QRob_StateMachine.State_complete;
END_TRANSITION
STEP sleep10:
END_STEP
TRANSITION FROM sleep10 TO Screw1H
    := sleep10.t > T#2s and not QRob_StateMachine.State_complete;
END_TRANSITION
STEP Screw1H:
    Screw1_entry(P1);  // entry action
    Screw1_active(N);  // step action
    Screw1_exit(P0);  // exit action
END_STEP
TRANSITION FROM Screw1H TO Open_gripkit
    := QRob_StateMachine.State_complete;
END_TRANSITION
STEP Open_gripkit:
END_STEP
TRANSITION FROM Open_gripkit TO Reset_ctr
    := read_bool_flag(True);
END_TRANSITION
STEP Reset_ctr:
    Reset_ctr_entry(P1);  // entry action
    Reset_ctr_active(N);  // step action
    Reset_ctr_exit(P0);  // exit action
END_STEP
TRANSITION FROM Reset_ctr TO sleep11
    := QRob_StateMachine.State_complete;
END_TRANSITION
STEP sleep11:
    sleep11_active(N);  // step action
    sleep11_exit(P0);  // exit action
END_STEP
TRANSITION FROM sleep11 TO Up_Robot_H
    := UR5_StateMachine.State_complete;
END_TRANSITION
STEP Up_Robot_H:
    Up_Robot_H_entry(P1);  // entry action
    Up_Robot_H_active(N);  // step action
    Up_Robot_H_exit(P0);  // exit action
END_STEP
TRANSITION FROM Up_Robot_H TO End_G10
    := UR5_StateMachine.State_complete;
END_TRANSITION
STEP End_G10:
    End_G10_exit(P0);  // exit action
END_STEP
TRANSITION FROM End_G10 TO Finish
    := true;
END_TRANSITION
TRANSITION FROM Inicio TO GState11
    := Global_state = 11;
END_TRANSITION
// macro Take_Buffer begins
STEP GState11:
END_STEP
TRANSITION FROM GState11 TO Qrob_Ctr_P_11
    := true;
END_TRANSITION
STEP Qrob_Ctr_P_11:
    Qrob_Ctr_P_entry(P1);  // entry action
    Qrob_Ctr_P_exit(P0);  // exit action
END_STEP
TRANSITION FROM Qrob_Ctr_P_11 TO sleepG11_1
    := QRob_StateMachine.State_complete;
END_TRANSITION
STEP sleepG11_1:
END_STEP
TRANSITION FROM sleepG11_1 TO take_buffer_11
    := sleepG11_1.t > T#2s;
END_TRANSITION
STEP take_buffer_11:
    take_buffer_11_entry(P1);  // entry action
    take_buufer_active(N);  // step action
END_STEP
TRANSITION FROM take_buffer_11 TO Qrob_Mov_AH
    := read_bool_flag(True);
END_TRANSITION
STEP Qrob_Mov_AH:
    Mov_AH_entry(P1);  // entry action
    Mov_AH_exit(P0);  // exit action
END_STEP
TRANSITION FROM Qrob_Mov_AH TO Wait_fin
    := QRob_StateMachine.State_complete;
END_TRANSITION
STEP Wait_fin:
    Wait_fin_active(N);  // step action
    Wait_fin_exit(P0);  // exit action
END_STEP
TRANSITION FROM Wait_fin TO End_G11
    := UR5_StateMachine.State_complete;
END_TRANSITION
STEP End_G11:
    End_G11_exit(P0);  // exit action
END_STEP
TRANSITION FROM End_G11 TO Finish
    := true;
END_TRANSITION
TRANSITION FROM Inicio TO GState12
    := Global_state = 12;
END_TRANSITION
// macro Cam2Up begins
STEP GState12:
END_STEP
TRANSITION FROM GState12 TO UR5Cam2Up
    := true;
END_TRANSITION
STEP UR5Cam2Up:
    UR5Cam2Up_entry(P1);  // entry action
    UR5Cam2Up_active(N);  // step action
    UR5Cam2Up_exit(P0);  // exit action
END_STEP
TRANSITION FROM UR5Cam2Up TO End_G12
    := UR5_StateMachine.State_complete;
END_TRANSITION
STEP End_G12:
    End_G12_exit(P0);  // exit action
END_STEP
TRANSITION FROM End_G12 TO Finish
    := true;
END_TRANSITION
TRANSITION FROM Inicio TO GState13
    := Global_state = 13;
END_TRANSITION
// macro Return_R begins
STEP GState13:
END_STEP
TRANSITION FROM GState13 TO (UR5_return, UR3_return)
    := true;
END_TRANSITION
STEP UR5_return:
    UR5_return_entry(P1);  // entry action
    UR5_return_active(N);  // step action
END_STEP
STEP UR3_return:
    UR3_return_entry(P1);  // entry action
    UR3_return_active(N);  // step action
END_STEP
TRANSITION FROM (UR5_return, UR3_return) TO End_G13
    := return_ur3 and return_ur5;
END_TRANSITION
STEP End_G13:
    End_G13_exit(P0);  // exit action
END_STEP
TRANSITION FROM End_G13 TO Finish
    := true;
END_TRANSITION
STEP Finish:
END_STEP
TRANSITION FROM Finish TO Wrt_FState
    := True;
END_TRANSITION
STEP Wrt_FState:
END_STEP
TRANSITION FROM Wrt_FState TO Init
    := Wrt_FState.t > T#100ms;
END_TRANSITION

ACTION Aux_active:
IF QRob_StateMachine.State_complete THEN
	qrob_home_flag := TRUE;
END_IF
END_ACTION

ACTION Aux_entry:
//Home Qrob Position
QRob_StateMachine.G_STATE := QrCts.MOVESTATE_HOME;
END_ACTION

ACTION Call_MaSta_active:
//cal UR3 state Machine
//UR3(init, state_to_exec,out_proces,out_global_state, out_internal_state
//IF User_Test_Sate <30 THEN
IF User_Test_Sate >0 AND User_Test_Sate <30 THEN
Vision_StateMachine.init_ := TRUE;
Vision_StateMachine.G_STATE := User_Test_Sate;
finish_state := Vision_StateMachine.State_complete;

//Vision_StateMachine(init_:=TRUE, G_STATE:=User_Test_Sate, State_complete=>finish_state,Act_Gl_State=>VisionRetVarState.Actual_GLV_State,Act_In_State=>VisionRetVarState.Actual_In_State);
//Vision_StateMachine(init_:=TRUE, G_STATE:=User_Test_Sate);
//finish_state:=Vision_StateMachine.State_complete;
//VisionRetVarState.Actual_GLV_State:=Vision_StateMachine.Act_Gl_State;
//VisionRetVarState.Actual_In_State:=Vision_StateMachine.Act_In_State;
ELSIF User_Test_Sate >=30 AND User_Test_Sate<50 THEN //UR3 States
UR3_StateMachine.init_ := TRUE;
UR3_StateMachine.G_STATE := User_Test_Sate;
finish_state := UR3_StateMachine.State_complete;

//UR3_StateMachine(init_:=TRUE, G_STATE:=User_Test_Sate, State_complete=>finish_state,Act_Gl_State=>UR3RetVarState.Actual_GLV_State,Act_In_State=>UR3RetVarState.Actual_In_State);	
//UR3_StateMachine(init_:=TRUE, G_STATE:=User_Test_Sate);
//finish_state:= UR3_StateMachine.State_complete;
//UR3RetVarState.Actual_GLV_State:=UR3_StateMachine.Act_Gl_State;
//UR3RetVarState.Actual_In_State:=UR3_StateMachine.Act_In_State;
ELSIF User_Test_Sate >=50 AND User_Test_Sate < 100THEN	//UR5 states
UR5_StateMachine.init_ := TRUE;
UR5_StateMachine.G_STATE := User_Test_Sate;
finish_state := UR5_StateMachine.State_complete;
UR5_StateMachine.Num_Ctr_Cam := cam_pos;
//UR5_StateMachine(init_:=TRUE, G_STATE:=User_Test_Sate, Num_Ctr_Cam:=-1,State_complete=>finish_state, Act_Gl_State=>UR5RetVarState.Actual_GLV_State,Act_In_State=>UR5RetVarState.Actual_In_State);	
//UR5_StateMachine(init_:=TRUE, G_STATE:=User_Test_Sate);
//finish_state:= UR5_StateMachine.State_complete;
//UR5RetVarState.Actual_GLV_State:=UR5_StateMachine.Act_Gl_State;
//UR5RetVarState.Actual_In_State:=UR5_StateMachine.Act_In_State;

ELSIF User_Test_Sate >=50 AND User_Test_Sate < 100THEN	//Qrob States
	//QRob_StateMachine(init_:=TRUE);
END_IF
END_ACTION

ACTION Call_MaSta_exit:
//reset satte variable
User_Test_Sate:=-1;
finish_state := False;
END_ACTION

ACTION Cam1UR5_active:

END_ACTION

ACTION Cam1UR5_entry:





UR5_StateMachine.G_STATE :=RCts.UR5Camera1;
//set cam position
cam_pos := 1;
END_ACTION

ACTION Cam1UR5_exit:

UR5_StateMachine.G_STATE := RCts.RESET_STATE;
END_ACTION

ACTION Catch_active:

END_ACTION

ACTION Catch_entry:
//call respective state to ur3 robot
//UR3_StateMachine(init_:=TRUE, G_STATE:=RCts.UR3CatchSeparator, State_complete=>UR3FinishState, Act_Gl_State=>UR3RetVarState.Actual_GLV_State,Act_In_State=>UR3RetVarState.Actual_In_State);

UR3_StateMachine.G_STATE := RCts.UR3CatchSeparator;
END_ACTION

ACTION Catch_exit_0:
//reset UR3
UR3_StateMachine.G_STATE := RCts.RESET_STATE;
END_ACTION

ACTION Ck_Eror_active:
IF QRob_StateMachine.State_complete THEN
	qrob_home_flag := TRUE;
END_IF
END_ACTION

ACTION Ck_Eror_entry:
//get struct values. cx, cy desviation from vision system 
IF cam_pos = 1 OR cam_pos =2 THEN
cx_vision_data := ck_real_value(Vision_struct.Cx_value_nut);
cy_vision_data := ck_real_value(Vision_struct.Cy_value_nut);
error_vision := 1.5;
ELSIF cam_pos = 3 OR cam_pos =4 THEN
cx_vision_data := ck_real_value(Vision_struct.Cx_value_hole);
cy_vision_data := ck_real_value(Vision_struct.Cy_value_hole);	
error_vision := 1.5;
END_IF	

//check is values are correct
IF cx_vision_data.Flag AND cy_vision_data.Flag THEN
	
	//Control Cam Position Ok
	IF ( ABS(cx_vision_data.Value) < error_vision) AND ( ABS(cy_vision_data.Value) < error_vision) THEN 
		Cam_center_ok := TRUE;
	ELSE 
		Cam_center_ok := FALSE;	
	END_IF
	
END_IF
END_ACTION

ACTION Ck_Eror_exit:

//reset var 
Cam_center_ok := False;
END_ACTION

ACTION Ck_Sep_pos_active:
//call respective state to machine system
//Vision_StateMachine(init_:=TRUE, G_STATE:=User_Test_Sate, State_complete=>finish_state,Act_Gl_State=>VisionRetVarState.Actual_GLV_State,Act_In_State=>VisionRetVarState.Actual_In_State);
END_ACTION

ACTION Crt_Pos_Cam1_active:
IF QRob_StateMachine.State_complete THEN
	qrob_home_flag := TRUE;
END_IF
END_ACTION

ACTION Crt_Pos_Cam1_entry:

IF cam_pos = 1 THEN 
	UR5_StateMachine.Num_Ctr_Cam := 1;
ELSIF cam_pos = 2 THEN
	UR5_StateMachine.Num_Ctr_Cam := 2;
ELSIF cam_pos = 3 THEN
	UR5_StateMachine.Num_Ctr_Cam := 3;
ELSIF cam_pos = 4 THEN
	UR5_StateMachine.Num_Ctr_Cam := 4;	
END_IF


UR5_StateMachine.G_STATE := RCts.UR5CtrCamPos;
END_ACTION

ACTION Crt_Pos_Cam1_exit:

UR5_StateMachine.G_STATE := RCts.RESET_STATE;
UR5_StateMachine.Num_Ctr_Cam := -1;
END_ACTION

ACTION Ctr_pos_entry:


//Change to Position Control 
QRob_StateMachine.G_STATE := QrCts.MOVESTATE_CTR_W;
QRob_StateMachine.Control := E_DRIVEOPERATIONMODE.DriveOperationMode_Pos1;
END_ACTION

ACTION Ctr_pos_exit:
//reset Qrob vars
QRob_StateMachine.G_STATE := -1;
write_bool_flag(FALSE);
END_ACTION

ACTION Ctr_pos_R_active:

END_ACTION

ACTION Ctr_pos_R_entry:
IF cam_pos = 1 THEN 
	UR5_StateMachine.G_STATE :=RCts.UR5CtrHeadTurnR;
	UR5_StateMachine.Num_Ctr_Cam := 1;
ELSIF cam_pos = 2 THEN
	UR5_StateMachine.G_STATE :=RCts.UR5CtrHeadTurnL;
	UR5_StateMachine.Num_Ctr_Cam := 2;
END_IF
END_ACTION

ACTION Ctr_pos_R_exit:

UR5_StateMachine.G_STATE := RCts.RESET_STATE;
END_ACTION

ACTION Ctr_posB_entry:


//Change to Position Control 
QRob_StateMachine.G_STATE := QrCts.MOVESTATE_CTR_W;
QRob_StateMachine.Control := E_DRIVEOPERATIONMODE.DriveOperationMode_Pos1;
END_ACTION

ACTION Ctr_posB_exit:
//reset Qrob vars
QRob_StateMachine.G_STATE := -1;
write_bool_flag(FALSE);
END_ACTION

ACTION Ctr_T_yaw_entry:
//Move Qrob to correct the offset between the screw and the axis

IF cam_pos = 1 OR cam_pos =2 THEN 
	nut_turn_data := ck_real_value(Vision_struct.Nut_turn_value);
	//home qrob while angle
	turn_aux_int := (REAL_TO_INT(Get_QRob_Pos.actual_position/360));
	turn_aux_float := INT_TO_REAL(turn_aux_int);
	turn_aux_float := -turn_aux_float  + (Get_QRob_Pos.actual_position/360);
	turn_aux_float := -1*(turn_aux_float*360);
	
	IF nut_turn_data.Flag = TRUE THEN
		QRob_StateMachine.Position := (Get_QRob_Pos.actual_position + turn_aux_float) + nut_turn_data.Value;
		QRob_StateMachine.Velocity := 100;
		QRob_StateMachine.G_STATE := QrCts.MOVESTATE_MOVABS;	
	END_IF

ELSIF 	cam_pos = 3 OR cam_pos =4 THEN 
	QRob_StateMachine.Position := 0;
	QRob_StateMachine.Velocity := 10;
	QRob_StateMachine.G_STATE := QrCts.MOVESTATE_MOVABS;	
END_IF
END_ACTION

ACTION Ctr_T_yaw_exit:
//reset Qrob vars
QRob_StateMachine.G_STATE := -1;
qrob_home_flag := FALSE;
END_ACTION

ACTION Ctr_Torque_active:

END_ACTION

ACTION Ctr_Torque_entry:

//change control to torque
QRob_StateMachine.G_STATE := QrCts.MOVESTATE_CTR_W;
QRob_StateMachine.Control := E_DRIVEOPERATIONMODE.DriveOperationMode_Torque;
END_ACTION

ACTION Ctr_Torque_exit:
//reset Qrob state
QRob_StateMachine.G_STATE := -1;
END_ACTION

ACTION Ctr_Torque1_entry:

//change control to torque
QRob_StateMachine.G_STATE := QrCts.MOVESTATE_CTR_W;
QRob_StateMachine.Control := E_DRIVEOPERATIONMODE.DriveOperationMode_Torque;
END_ACTION

ACTION Ctr_Torque1_exit:
//reset Qrob state
QRob_StateMachine.G_STATE := -1;
END_ACTION

ACTION DropBench_active:

END_ACTION

ACTION DropBench_entry:


UR3_StateMachine.G_STATE :=RCts.UR3DropBench;
END_ACTION

ACTION DropBench_exit:

UR3_StateMachine.G_STATE := RCts.RESET_STATE;
END_ACTION

ACTION End_6_exit:
IF cam_pos = 1 THEN 
	Global_State := 6; 
ELSIF cam_pos = 2 THEN
	Global_State := 6; 
ELSIF cam_pos = 3 THEN
	Global_State := 10; 
ELSIF cam_pos = 4 THEN
	Global_State := 10; 
END_IF
END_ACTION

ACTION End_8_exit:

IF cam_pos = 1 THEN 
	Global_State  := 7;
ELSIF cam_pos = 2 THEN 
	Global_State := 9;
END_IF
END_ACTION

ACTION End_9_exit:

Global_State := 8;
END_ACTION

ACTION End_exit:
Global_State := 5;
END_ACTION

ACTION End_G1_exit:

//next state
Global_State := 2;
//actual cam position
cam_pos := 1;
END_ACTION

ACTION End_G10_exit:
IF cam_pos = 3 THEN 
Global_State := 11; 
write_bool_flag(FALSE);
ELSIF cam_pos = 4 THEN 
Global_State := 13; 	
END_IF
END_ACTION

ACTION End_G11_exit:
Global_State := 12;
cam_pos := 4;
END_ACTION

ACTION End_G12_exit:

cam_pos := 4;
Global_State := 5;
END_ACTION

ACTION End_G13_exit:
Global_State := -1;
cam_pos := -1;

return_ur5 := FALSE;;
return_ur3 := FALSE;
END_ACTION

ACTION End_G7_exit:
Global_State := 8;
END_ACTION

ACTION End_G8_exit:
cam_pos := 2;
Global_State := 3;
END_ACTION

ACTION End_G9_exit:
cam_pos := 3;
Global_State := 5;
END_ACTION

ACTION Finish_s2_exit_0:
sep_pos_data := ck_real_value(Vision_struct.Pos_sep);

IF  sep_pos_data.Value = VCts.Separador_correct THEN
	//separator correct position
	Global_State := 3;
	//set cam_pos to indicate work on firts camera
	cam_pos := 1;
ELSIF sep_pos_data.Value = VCts.Separador_turned THEN
	//separator wrong position
	//Global_State := 4;
	Global_State := 3;
	//set cam_pos to indicate work on firts camera
	cam_pos := 1;
END_IF
END_ACTION

ACTION Force_down_active:

END_ACTION

ACTION GState10_exit:
//set setpoint torque 
Torque_SetPoint := 600;
END_ACTION

ACTION GState7_exit:
//set setpoint torque 
Torque_SetPoint := 70;
END_ACTION

ACTION Iniciar_entry:

//init the machines States
Vision_StateMachine.init_ := TRUE;
UR3_StateMachine.init_ := TRUE;
UR5_StateMachine.init_ := TRUE;
QRob_StateMachine.init_ := TRUE;
END_ACTION

ACTION Mov_AH_entry:
QRob_StateMachine.Position := Get_QRob_Pos.actual_position -(4*360);
QRob_StateMachine.Velocity := 50;
QRob_StateMachine.G_STATE := QrCts.MOVESTATE_MOVABS;
END_ACTION

ACTION Mov_AH_exit:
write_bool_flag(True);
END_ACTION

ACTION Move_S_entry:

UR3_StateMachine.G_STATE := RCts.UR3Move;
END_ACTION

ACTION Move_S_exit:
//reset UR3
UR3_StateMachine.G_STATE := RCts.RESET_STATE;
END_ACTION

ACTION Move_to_buffer_active:

END_ACTION

ACTION Move_to_buffer_entry:
UR5_StateMachine.G_STATE := RCts.UR5DropHead;
UR5_StateMachine.Num_Ctr_Cam := -1;
END_ACTION

ACTION Move_to_buffer_exit:
UR5_StateMachine.G_STATE := RCts.RESET_STATE;
UR5_StateMachine.Num_Ctr_Cam := -1;
END_ACTION

ACTION Move_to_Nut_active:
ck_operation := read_bool_flag(True);
END_ACTION

ACTION Move_to_Nut_entry:
IF cam_pos = 1 THEN 
	UR5_StateMachine.Num_Ctr_Cam := 1;
ELSIF cam_pos = 2 THEN
	UR5_StateMachine.Num_Ctr_Cam := 2;
ELSIF cam_pos = 3 THEN
	UR5_StateMachine.Num_Ctr_Cam := 3;
ELSIF cam_pos = 4 THEN
	UR5_StateMachine.Num_Ctr_Cam := 4;
END_IF


UR5_StateMachine.G_STATE := RCts.UR5MoveToNut;
UR3_StateMachine.G_STATE := RCts.UR3Correct_Insertion;
END_ACTION

ACTION Move_to_Nut_exit:
UR5_StateMachine.G_STATE := RCts.RESET_STATE;
UR5_StateMachine.Num_Ctr_Cam := -1;
END_ACTION

ACTION MoveS_active:

END_ACTION

ACTION MOVESEP_exit:
//changet the state to exec
STATE := RCts.UR3CatchSeparator;
END_ACTION

ACTION Mv_robot_up_active:

//read force from Ur3 and send to Ur5
wr_real_value(RCts.UR_DATA_SEND,flip_byte(Robot_UR3.UR_TCP.FLOAT14));
ck_operation := read_bool_flag(True);
END_ACTION

ACTION Nut_insert_active:
IF read_bool_flag(TRUE) THEN 
	UR3_StateMachine.G_STATE := RCts.UR3Correct_Insertion;
END_IF
END_ACTION

ACTION Nut_insert_entry:
//set to zero Ur3 forze sensor
UR3_StateMachine.G_STATE := RCts.UR3Correct_Insertion;

QRob_StateMachine.Position := Get_QRob_Pos.actual_position -(10*360);
//QRob_StateMachine.Position := QRob_StateMachine.Act_Pos -(10*360);
QRob_StateMachine.Velocity := 5;
QRob_StateMachine.G_STATE := QrCts.MOVESTATE_MOVABS;	


UR5_StateMachine.G_STATE := RCts.UR5Correct_Insertion;
ck_operation := FALSE;
END_ACTION

ACTION Nut_insert_exit:
UR5_StateMachine.G_STATE := RCts.RESET_STATE;
UR5_StateMachine.Num_Ctr_Cam := -1;
END_ACTION

ACTION Pic_left_active:
Vision_StateMachine.init_:= TRUE;
Vision_StateMachine.G_STATE := VCts.SeparatorRot_L;
END_ACTION

ACTION Pic_left_exit:
Vision_StateMachine.init_ := FALSE;
Vision_StateMachine.G_STATE := VCts.RESET;
END_ACTION

ACTION Pic_rigth_active:

END_ACTION

ACTION Pic_rigth_entry:


//select state according to robot position 
IF cam_pos = 1 THEN 
	Vision_StateMachine.G_STATE := VCts.SeparatorRot_R;
ELSIF cam_pos = 2 THEN
	Vision_StateMachine.G_STATE := VCts.SeparatorRot_L;
END_IF
END_ACTION

ACTION Pic_rigth_exit:

Vision_StateMachine.G_STATE := VCts.RESET;
END_ACTION

ACTION Pos_Sep_active:

END_ACTION

ACTION Pos_Sep_entry:

UR5_StateMachine.G_STATE :=RCts.UR5CkPosSepator;
END_ACTION

ACTION Pos_Sep_exit:

UR5_StateMachine.G_STATE := RCts.RESET_STATE;
END_ACTION

ACTION Qrob_Ctr_P_entry:


//Change to Position Control 
QRob_StateMachine.G_STATE := QrCts.MOVESTATE_CTR_W;
QRob_StateMachine.Control := E_DRIVEOPERATIONMODE.DriveOperationMode_Pos1;
END_ACTION

ACTION Qrob_Ctr_P_exit:
//reset Qrob vars
QRob_StateMachine.G_STATE := -1;
END_ACTION

ACTION Qrob_home_active:
IF QRob_StateMachine.State_complete THEN
	qrob_home_flag := TRUE;
END_IF
END_ACTION

ACTION Qrob_home_entry:

END_ACTION

ACTION Qrob_home_exit:

END_ACTION

ACTION Qrob_safe_entry:

QRob_StateMachine.Position := Get_QRob_Pos.actual_position -(3*360);
QRob_StateMachine.Velocity := 170;
QRob_StateMachine.G_STATE := QrCts.MOVESTATE_MOVABS;
END_ACTION

ACTION Qrob_safe_exit:

END_ACTION

ACTION Qrob_unSc_active:

END_ACTION

ACTION Qrob_unSc_entry:

//reset flag to indicate whwen qrob finish
write_bool_flag(FALSE);

//QRob_StateMachine.Position := Get_QRob_Pos.actual_position -(15*360);
//QRob_StateMachine.Position := QRob_StateMachine.Act_Pos -(15*360);
QRob_StateMachine.Position := (Global_servo.Axis1.NcToPlc.ActPos) -(12*360);
QRob_StateMachine.Velocity := 170;
QRob_StateMachine.G_STATE := QrCts.MOVESTATE_MOVABS;	


UR5_StateMachine.Num_Ctr_Cam := -1;	
UR5_StateMachine.G_STATE := RCts.UR5UnScrew;
END_ACTION

ACTION Qrob_unSc_exit:

//reset Qrob vars
QRob_StateMachine.G_STATE := -1;
//set to indicate qrob_finish
write_bool_flag(TRUE);
END_ACTION

ACTION Qrob_unSc1_entry:

//reset flag to indicate whwen qrob finish
write_bool_flag(FALSE);
//QRob_StateMachine.Position := (Get_QRob_Pos.actual_position) -(15*360);
//QRob_StateMachine.Position := QRob_StateMachine.Act_Pos -(15*360);

QRob_StateMachine.Position := (Global_servo.Axis1.NcToPlc.ActPos) -(12*360);
QRob_StateMachine.Velocity := 170;
QRob_StateMachine.G_STATE := QrCts.MOVESTATE_MOVABS;	


UR5_StateMachine.Num_Ctr_Cam := -1;	
UR5_StateMachine.G_STATE := RCts.UR5UnScrew;
END_ACTION

ACTION Qrob_unSc1_exit:

//reset Qrob vars
QRob_StateMachine.G_STATE := -1;
//set to indicate qrob_finish
write_bool_flag(TRUE);

//set to zero Ur3 forze sensor
UR3_StateMachine.G_STATE := RCts.UR3Correct_Insertion;
END_ACTION

ACTION Qrob_unSc2_active:
//read force from Ur3 and send to Ur5
wr_real_value(RCts.UR_DATA_SEND,flip_byte(Robot_UR3.UR_TCP.FLOAT14));
END_ACTION

ACTION Qrob_unSc2_entry:

//reset flag to indicate whwen qrob finish
write_bool_flag(FALSE);
//QRob_StateMachine.Position := (Get_QRob_Pos.actual_position) -(15*360);
//QRob_StateMachine.Position := QRob_StateMachine.Act_Pos -(15*360);

QRob_StateMachine.Position := (Global_servo.Axis1.NcToPlc.ActPos) -(10*360);
QRob_StateMachine.Velocity := 120;
QRob_StateMachine.G_STATE := QrCts.MOVESTATE_MOVABS;	


UR5_StateMachine.Num_Ctr_Cam := -1;	
UR5_StateMachine.G_STATE := RCts.UR5UnScrew;
END_ACTION

ACTION Qrob_unSc2_exit:
//reset Qrob vars
QRob_StateMachine.G_STATE := -1;
//set to indicate qrob_finish
END_ACTION

ACTION Relief_entry:


//reset torque state to relive the remant torques.
QRob_StateMachine.G_STATE := QrCts.MOVESTATE_RESET;
END_ACTION

ACTION Relief_exit:
//reset Qrob state
QRob_StateMachine.G_STATE := -1;
END_ACTION

ACTION Reset_ctr_active:

END_ACTION

ACTION Reset_ctr_entry:
//reset torque state to relive the remant torques.
QRob_StateMachine.G_STATE := QrCts.MOVESTATE_RESET;
write_bool_flag(False);
END_ACTION

ACTION Reset_ctr_exit:
//reset Qrob state
QRob_StateMachine.G_STATE := -1;
screw_finish := FALSE;
END_ACTION

ACTION reset_entry:

//reset torque state to relive the remant torques.
QRob_StateMachine.G_STATE := QrCts.MOVESTATE_RESET;
write_bool_flag(False);
END_ACTION

ACTION reset_exit:


//reset Qrob state
QRob_StateMachine.G_STATE := -1;
END_ACTION

ACTION Reset_force_entry:
//set to zero Ur3 forze sensor
UR3_StateMachine.G_STATE := RCts.UR3Correct_Insertion;
END_ACTION

ACTION Reset_force_exit:
UR3_StateMachine.G_STATE := RCts.RESET_STATE;
END_ACTION

ACTION Reset_Qrob_active:

END_ACTION

ACTION Reset_Qrob_entry:
// NETWORK 1
END_ACTION

ACTION Reset_Qrob_entry_0:
//stop Qrob 
QRob_StateMachine.Reset_state := TRUE;
END_ACTION

ACTION Reset_Qrob_exit:
//reset Qrob vars
QRob_StateMachine.G_STATE := -1;
END_ACTION

ACTION Reset_Qrob2_entry:

//reset torque state to relive the remant torques.
QRob_StateMachine.G_STATE := QrCts.MOVESTATE_RESET;
END_ACTION

ACTION Reset_Qrob2_exit:
//reset Qrob state
QRob_StateMachine.G_STATE := -1;
END_ACTION

ACTION Robot_up_active:

END_ACTION

ACTION Robot_up_exit:
UR5_StateMachine.G_STATE := RCts.RESET_STATE;
UR5_StateMachine.Num_Ctr_Cam := -1;


QRob_StateMachine.G_STATE := -1;
//reset bool flags 
write_bool_flag(FALSE);
END_ACTION

ACTION ScB_active:

END_ACTION

ACTION ScB_entry:
QRob_StateMachine.Torque := Torque_SetPoint;
QRob_StateMachine.Velocity := 100;
QRob_StateMachine.Torque_ramp := 200;
//iniacialize torque state.
QRob_StateMachine.G_STATE := QrCts.MOVESTATE_TORQUE;
END_ACTION

ACTION ScB_exit:
//reset Qrob state
QRob_StateMachine.G_STATE := -1;
write_bool_flag(TRUE);
END_ACTION

ACTION Screw_F_active:
IF UR5_StateMachine.State_complete THEN 
	screw_finish := TRUE;
END_IF
END_ACTION

ACTION Screw_F_entry:

END_ACTION

ACTION Screw_F_exit:
UR5_StateMachine.G_STATE := RCts.RESET_STATE;
UR5_StateMachine.Num_Ctr_Cam := -1;
END_ACTION

ACTION Screw_finish_active:
IF UR5_StateMachine.State_complete = TRUE THEN 
	screw_finish := TRUE;
END_IF
END_ACTION

ACTION Screw_finish_exit:
UR5_StateMachine.G_STATE := RCts.RESET_STATE;
UR5_StateMachine.Num_Ctr_Cam := -1;
END_ACTION

ACTION Screw1_active:

END_ACTION

ACTION Screw1_entry:



QRob_StateMachine.Torque := Torque_SetPoint;
QRob_StateMachine.Velocity := 100;
QRob_StateMachine.Torque_ramp := 200;
//iniacialize torque state.
QRob_StateMachine.G_STATE := QrCts.MOVESTATE_TORQUE;



UR5_StateMachine.G_STATE := RCts.UR5ScrewHigh;
END_ACTION

ACTION Screw1_exit:
//reset Qrob state
QRob_StateMachine.G_STATE := -1;
write_bool_flag(TRUE);
END_ACTION

ACTION Screw1B_entry:
QRob_StateMachine.Torque := Torque_SetPoint;
QRob_StateMachine.Velocity := 100;
QRob_StateMachine.Torque_ramp := 200;
//iniacialize torque state.
QRob_StateMachine.G_STATE := QrCts.MOVESTATE_TORQUE;
END_ACTION

ACTION Screw1B_exit:
//reset Qrob state
QRob_StateMachine.G_STATE := -1;
write_bool_flag(TRUE);
END_ACTION

ACTION ScrewBuff_active:

END_ACTION

ACTION ScrewBuff_entry:

UR5_StateMachine.G_STATE := RCts.UR5Screw;	
UR5_StateMachine.Num_Ctr_Cam := -1;
END_ACTION

ACTION Set_Ctr_entry:

//change control to torque
QRob_StateMachine.G_STATE := QrCts.MOVESTATE_CTR_W;
QRob_StateMachine.Control := E_DRIVEOPERATIONMODE.DriveOperationMode_Torque;
END_ACTION

ACTION Set_Ctr_exit:
//reset Qrob state
QRob_StateMachine.G_STATE := -1;
END_ACTION

ACTION sleep11_active:

END_ACTION

ACTION sleep11_entry:
UR5_StateMachine.G_STATE := RCts.RESET_STATE;
UR5_StateMachine.Num_Ctr_Cam := -1;
END_ACTION

ACTION sleep11_entry_0:

END_ACTION

ACTION sleep11_exit:



UR5_StateMachine.G_STATE := RCts.RESET_STATE;
UR5_StateMachine.Num_Ctr_Cam := -1;
write_bool_flag(FALSE);
END_ACTION

ACTION sleep12_exit:
write_bool_flag(False);
END_ACTION

ACTION sleep6_10_active:
//read force from Ur3 and send to Ur5
wr_real_value(RCts.UR_DATA_SEND,flip_byte(Robot_UR3.UR_TCP.FLOAT14));
ck_operation := read_bool_flag(True);
END_ACTION

ACTION sleepS7_exit:

END_ACTION

ACTION Stop_qrob_entry:
//stop Qrob 
QRob_StateMachine.Reset_state := TRUE;
END_ACTION

ACTION Stop_qrob_exit:
//reset Qrob vars
QRob_StateMachine.G_STATE := -1;
END_ACTION

ACTION take_buffer_11_entry:
UR5_StateMachine.G_STATE := RCts.UR5TakeBuffer;
END_ACTION

ACTION take_buufer_active:

END_ACTION

ACTION take_buufer_exit:

END_ACTION

ACTION Take_Pic_active:

END_ACTION

ACTION Take_Pic_entry:

//Vision_StateMachine.G_STATE := VCts.SeparatorPos;
Vision_StateMachine.G_STATE := VCts.SeparatorPos;
END_ACTION

ACTION Take_Pic_exit:


Vision_StateMachine.G_STATE := VCts.RESET;
END_ACTION

ACTION Take_Pic1_active:
IF QRob_StateMachine.State_complete THEN
	qrob_home_flag := TRUE;
END_IF
END_ACTION

ACTION Take_Pic1_entry:
IF cam_pos = 1 OR cam_pos= 2 THEN
	Vision_StateMachine.G_STATE := VCts.SeparatorNut;
ELSIF 	cam_pos = 3 OR cam_pos= 4 THEN
	Vision_StateMachine.G_STATE := VCts.SeparatorHole;	
END_IF
END_ACTION

ACTION Take_Pic1_exit:
Vision_StateMachine.G_STATE := VCts.RESET;
END_ACTION

ACTION Turn_relief_entry:


screw_finish := FALSE;
QRob_StateMachine.Position := Get_QRob_Pos.actual_position  - 2;
QRob_StateMachine.Velocity := 50;
QRob_StateMachine.G_STATE := QrCts.MOVESTATE_MOVABS;
END_ACTION

ACTION Turn_relief_exit:
//reset Qrob vars
QRob_StateMachine.G_STATE := -1;
END_ACTION

ACTION UnScrew_7_active:

END_ACTION

ACTION UnScrew_7_entry:


//change control to torque
QRob_StateMachine.G_STATE := QrCts.MOVESTATE_CTR_W;
QRob_StateMachine.Control := E_DRIVEOPERATIONMODE.DriveOperationMode_Pos1;
END_ACTION

ACTION UnScrew_7_exit:
QRob_StateMachine.G_STATE := -1;
END_ACTION

ACTION Up_Robot_active:

END_ACTION

ACTION Up_Robot_entry:
UR5_StateMachine.G_STATE := RCts.UR5UpRobotAs;
UR5_StateMachine.Num_Ctr_Cam := -1;
END_ACTION

ACTION Up_Robot_exit:
UR5_StateMachine.G_STATE := RCts.RESET_STATE;
UR5_StateMachine.Num_Ctr_Cam := -1;
END_ACTION

ACTION Up_Robot_H_active:

END_ACTION

ACTION Up_Robot_H_entry:
UR5_StateMachine.G_STATE := RCts.UR5UpRobotAs;
UR5_StateMachine.Num_Ctr_Cam := -1;
END_ACTION

ACTION Up_Robot_H_exit:
UR5_StateMachine.G_STATE := RCts.RESET_STATE;
UR5_StateMachine.Num_Ctr_Cam := -1;
screw_finish := FALSE;
write_bool_flag(FALSE);
END_ACTION

ACTION UR3_return_active:



IF UR3_StateMachine.State_complete THEN 
	return_ur3 := TRUE;
END_IF
END_ACTION

ACTION UR3_return_entry:
UR3_StateMachine.G_STATE := RCts.UR3Return;
END_ACTION

ACTION UR3UP_active:

END_ACTION

ACTION UR3UP_entry:

UR3_StateMachine.G_STATE := RCts.UR3DropCable;
END_ACTION

ACTION UR3UP_exit:

UR3_StateMachine.G_STATE := RCts.RESET_STATE;
END_ACTION

ACTION UR5_P_Cam_active:

END_ACTION

ACTION UR5_P_Cam_entry:
UR5_StateMachine.G_STATE := RCts.UR5Camera2;
UR5_StateMachine.Num_Ctr_Cam := -1;
END_ACTION

ACTION UR5_P_Cam_exit:
UR5_StateMachine.G_STATE := RCts.RESET_STATE;
UR5_StateMachine.Num_Ctr_Cam := -1;
END_ACTION

ACTION UR5_return_active:







IF UR5_StateMachine.State_complete THEN 
	return_ur5 := TRUE;
END_IF
END_ACTION

ACTION UR5_return_entry:
UR5_StateMachine.G_STATE := RCts.UR5Return;
END_ACTION

ACTION UR5_scre_f_exit:
UR5_StateMachine.G_STATE := RCts.RESET_STATE;
UR5_StateMachine.Num_Ctr_Cam := -1;
END_ACTION

ACTION UR5_UP_C1_active:

END_ACTION

ACTION UR5_UP_C1_entry:
UR5_StateMachine.G_STATE := RCts.UR5UpCamera1;
UR5_StateMachine.Num_Ctr_Cam := -1;
END_ACTION

ACTION UR5_UP_C1_exit:
UR5_StateMachine.Num_Ctr_Cam := -1;
END_ACTION

ACTION UR5Cam2Up_active:

END_ACTION

ACTION UR5Cam2Up_entry:
UR5_StateMachine.G_STATE := RCts.UR5UpCamera2;
END_ACTION

ACTION UR5Cam2Up_exit:
UR5_StateMachine.G_STATE := RCts.RESET_STATE;
END_ACTION

ACTION Wait_fin_active:

END_ACTION

ACTION Wait_fin_exit:
UR5_StateMachine.G_STATE := RCts.RESET_STATE;
END_ACTION

END_PROGRAM

// ---- POUs/POUs/ROBOTS/Robot_machine_state/UR3_StateMachine.TcPOU
PROGRAM UR3_StateMachine

VAR_INPUT
	init_: BOOL:= FALSE;
	G_STATE: INT:=-1;

END_VAR


VAR
	//internal aux state
	I_STATE : INT:=-1;
	
	//vars to start and stop Robot, safety segurity, power on
	UR3_Safety_pin_1 AT%Q*:BOOL:= FALSE;
	UR3_Safety_pin_2 AT%Q*:BOOL:= FALSE;
	UR3_Power_on AT%Q*:BOOL:= FALSE;
	UR3_Run_Robot AT%Q*:BOOL:= FALSE;
	
END_VAR


VAR_OUTPUT
	State_complete : BOOL:= FALSE;
	Act_Gl_State :INT:=-1;
	Act_In_State: INT:=-1;
END_VAR

VAR CONSTANT 
	

	
END_VAR

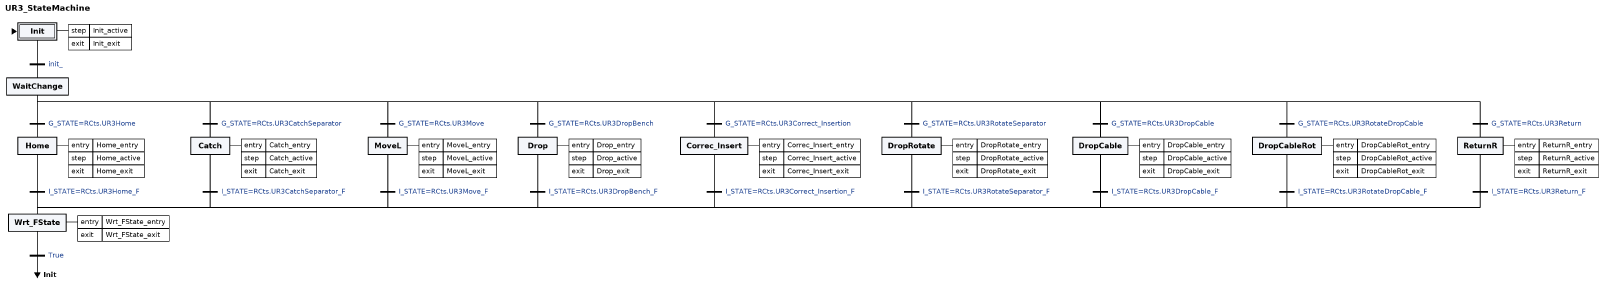
INITIAL_STEP Init:
    Init_active(N);  // step action
    Init_exit(P0);  // exit action
END_STEP
TRANSITION FROM Init TO WaitChange
    := init_;
END_TRANSITION
STEP WaitChange:
END_STEP
TRANSITION FROM WaitChange TO Home
    := G_STATE=RCts.UR3Home;
END_TRANSITION
STEP Home:
    Home_entry(P1);  // entry action
    Home_active(N);  // step action
    Home_exit(P0);  // exit action
END_STEP
TRANSITION FROM Home TO Wrt_FState
    := I_STATE=RCts.UR3Home_F;
END_TRANSITION
TRANSITION FROM WaitChange TO Catch
    := G_STATE=RCts.UR3CatchSeparator;
END_TRANSITION
STEP Catch:
    Catch_entry(P1);  // entry action
    Catch_active(N);  // step action
    Catch_exit(P0);  // exit action
END_STEP
TRANSITION FROM Catch TO Wrt_FState
    := I_STATE=RCts.UR3CatchSeparator_F;
END_TRANSITION
TRANSITION FROM WaitChange TO MoveL
    := G_STATE=RCts.UR3Move;
END_TRANSITION
STEP MoveL:
    MoveL_entry(P1);  // entry action
    MoveL_active(N);  // step action
    MoveL_exit(P0);  // exit action
END_STEP
TRANSITION FROM MoveL TO Wrt_FState
    := I_STATE=RCts.UR3Move_F;
END_TRANSITION
TRANSITION FROM WaitChange TO Drop
    := G_STATE=RCts.UR3DropBench;
END_TRANSITION
STEP Drop:
    Drop_entry(P1);  // entry action
    Drop_active(N);  // step action
    Drop_exit(P0);  // exit action
END_STEP
TRANSITION FROM Drop TO Wrt_FState
    := I_STATE=RCts.UR3DropBench_F;
END_TRANSITION
TRANSITION FROM WaitChange TO Correc_Insert
    := G_STATE=RCts.UR3Correct_Insertion;
END_TRANSITION
STEP Correc_Insert:
    Correc_Insert_entry(P1);  // entry action
    Correc_Insert_active(N);  // step action
    Correc_Insert_exit(P0);  // exit action
END_STEP
TRANSITION FROM Correc_Insert TO Wrt_FState
    := I_STATE=RCts.UR3Correct_Insertion_F;
END_TRANSITION
TRANSITION FROM WaitChange TO DropRotate
    := G_STATE=RCts.UR3RotateSeparator;
END_TRANSITION
STEP DropRotate:
    DropRotate_entry(P1);  // entry action
    DropRotate_active(N);  // step action
    DropRotate_exit(P0);  // exit action
END_STEP
TRANSITION FROM DropRotate TO Wrt_FState
    := I_STATE=RCts.UR3RotateSeparator_F;
END_TRANSITION
TRANSITION FROM WaitChange TO DropCable
    := G_STATE=RCts.UR3DropCable;
END_TRANSITION
STEP DropCable:
    DropCable_entry(P1);  // entry action
    DropCable_active(N);  // step action
    DropCable_exit(P0);  // exit action
END_STEP
TRANSITION FROM DropCable TO Wrt_FState
    := I_STATE=RCts.UR3DropCable_F;
END_TRANSITION
TRANSITION FROM WaitChange TO DropCableRot
    := G_STATE=RCts.UR3RotateDropCable;
END_TRANSITION
STEP DropCableRot:
    DropCableRot_entry(P1);  // entry action
    DropCableRot_active(N);  // step action
    DropCableRot_exit(P0);  // exit action
END_STEP
TRANSITION FROM DropCableRot TO Wrt_FState
    := I_STATE=RCts.UR3RotateDropCable_F;
END_TRANSITION
TRANSITION FROM WaitChange TO ReturnR
    := G_STATE=RCts.UR3Return;
END_TRANSITION
STEP ReturnR:
    ReturnR_entry(P1);  // entry action
    ReturnR_active(N);  // step action
    ReturnR_exit(P0);  // exit action
END_STEP
TRANSITION FROM ReturnR TO Wrt_FState
    := I_STATE=RCts.UR3Return_F;
END_TRANSITION
STEP Wrt_FState:
    Wrt_FState_entry(P1);  // entry action
    Wrt_FState_exit(P0);  // exit action
END_STEP
TRANSITION FROM Wrt_FState TO Init
    := True;
END_TRANSITION

ACTION Catch_active:
//read register from robot and chek is can read 2 or more correct values 
IF ck_state(RCts.UR3,RCts.UR3CatchSeparator_I) THEN
	 I_STATE:= RCts.UR3CatchSeparator_I;
ELSIF ck_state(RCts.UR3,RCts.UR3CatchSeparator_F) THEN
	I_STATE := RCts.UR3CatchSeparator_F;
END_IF

//read internal variable and write over output variable
Act_In_State := I_STATE;
END_ACTION

ACTION Catch_entry:
//write state variables to robot, to execute respective state.
wr_state(RCts.UR3,RCts.UR3CatchSeparator);
//write the retain state variable 
Act_Gl_State:=RCts.UR3CatchSeparator;
END_ACTION

ACTION Catch_exit:
//write reset state variables to robot.
wr_state(RCts.UR3,RCts.RESET_STATE);
//reset Global state variable
G_STATE := -1;
END_ACTION

ACTION Correc_Insert_active:
//read register from robot and chek is can read 2 or more correct values 
IF ck_state(RCts.UR3,RCts.UR3Correct_Insertion_I) THEN
	 I_STATE:= RCts.UR3Correct_Insertion_I;
ELSIF ck_state(RCts.UR3,RCts.UR3Correct_Insertion_F) THEN
	I_STATE := RCts.UR3Correct_Insertion_F;
END_IF


//read internal variable and write over output variable
Act_In_State := I_STATE;
END_ACTION

ACTION Correc_Insert_entry:
//write state variables to robot, to execute respective state.
wr_state(RCts.UR3,RCts.UR3Correct_Insertion);
//write the retain state variable 
Act_Gl_State:=RCts.UR3Correct_Insertion;
END_ACTION

ACTION Correc_Insert_exit:
//write reset state variables to robot.
wr_state(RCts.UR3,RCts.RESET_STATE);
//Assign a value according to the variable UserState
//-1 or respective NEXT state  CS.UR3DropBench
//wr_GL_STATE(CS.UR5Camera1,UserState);

//reset Global state variable
G_STATE := -1;
END_ACTION

ACTION Drop_active:
//read register from robot and chek is can read 2 or more correct values 
IF ck_state(RCts.UR3,RCts.UR3DropBench_I) THEN
	 I_STATE:= RCts.UR3DropBench_I;
ELSIF ck_state(RCts.UR3,RCts.UR3DropBench_F) THEN
	I_STATE := RCts.UR3DropBench_F;
END_IF


//read internal variable and write over output variable
Act_In_State := I_STATE;
END_ACTION

ACTION Drop_entry:
//write state variables to robot, to execute respective state.
wr_state(RCts.UR3,RCts.UR3DropBench);
//write the retain state variable 
Act_Gl_State:=RCts.UR3DropBench;
END_ACTION

ACTION Drop_exit:
//write reset state variables to robot.
wr_state(RCts.UR3,RCts.RESET_STATE);
//Assign a value according to the variable UserState
//-1 or respective NEXT state  CS.UR3DropBench
//wr_GL_STATE(CS.UR5Camera1,UserState);

//reset Global state variable
G_STATE := -1;
END_ACTION

ACTION DropCable_active:
//read register from robot and chek is can read 2 or more correct values 
IF ck_state(RCts.UR3,RCts.UR3DropCable_I) THEN
	 I_STATE:= RCts.UR3DropCable_I;
ELSIF ck_state(RCts.UR3,RCts.UR3DropCable_F) THEN
	I_STATE := RCts.UR3DropCable_F;
END_IF

//read internal variable and write over output variable
Act_In_State := I_STATE;
END_ACTION

ACTION DropCable_entry:
//write state variables to robot, to execute respective state.
wr_state(RCts.UR3,RCts.UR3DropCable);
//write the retain state variable 
Act_Gl_State:=RCts.UR3DropCable;
END_ACTION

ACTION DropCable_exit:
//write reset state variables to robot.
wr_state(RCts.UR3,RCts.RESET_STATE);
//reset Global state variable
G_STATE := -1;
END_ACTION

ACTION DropCableRot_active:
//read register from robot and chek is can read 2 or more correct values 
IF ck_state(RCts.UR3,RCts.UR3RotateDropCable_I) THEN
	 I_STATE:= RCts.UR3RotateDropCable_I;
ELSIF ck_state(RCts.UR3,RCts.UR3RotateDropCable_F) THEN
	I_STATE := RCts.UR3RotateDropCable_F;
END_IF


//read internal variable and write over output variable
Act_In_State := I_STATE;
END_ACTION

ACTION DropCableRot_entry:
//write state variables to robot, to execute respective state.
wr_state(RCts.UR3,RCts.UR3RotateDropCable);
//write the retain state variable 
Act_Gl_State:=RCts.UR3RotateDropCable;
END_ACTION

ACTION DropCableRot_exit:
//write reset state variables to robot.
wr_state(RCts.UR3,RCts.RESET_STATE);
//reset Global state variable
G_STATE := -1;
END_ACTION

ACTION DropRotate_active:

//read register from robot and chek is can read 2 or more correct values 
IF ck_state(RCts.UR3,RCts.UR3RotateSeparator_I) THEN
	 I_STATE:= RCts.UR3RotateSeparator_I;
ELSIF ck_state(RCts.UR3,RCts.UR3RotateSeparator_F) THEN
	I_STATE := RCts.UR3RotateSeparator_F;
END_IF

//read internal variable and write over output variable
Act_In_State := I_STATE;
END_ACTION

ACTION DropRotate_entry:
//write state variables to robot, to execute respective state.
wr_state(RCts.UR3,RCts.UR3RotateSeparator);
//write the retain state variable 
Act_Gl_State:=RCts.UR3RotateSeparator;
END_ACTION

ACTION DropRotate_exit:
//write reset state variables to robot.
wr_state(RCts.UR3,RCts.RESET_STATE);
//reset Global state variable
G_STATE := -1;
END_ACTION

ACTION Home_active:
//read register from robot and chek is can read 2 or more correct values 
IF ck_state(RCts.UR3,RCts.UR3Home_I) THEN
	 I_STATE:= RCts.UR3Home_I;
ELSIF ck_state(RCts.UR3,RCts.UR3Home_F) THEN
	I_STATE := RCts.UR3Home_F;
END_IF

//read internal variable and write over output variable
Act_In_State := I_STATE;
END_ACTION

ACTION Home_entry:
//write state variables to robot, to execute respective state.
wr_state(RCts.UR3,RCts.UR3Home);
//write the retain state variable 
Act_Gl_State:=RCts.UR3Home;
END_ACTION

ACTION Home_exit:
//write reset state variables to robot.
wr_state(RCts.UR3,RCts.RESET_STATE);
//reset Global state variable
G_STATE := -1;
END_ACTION

ACTION Init_active:

END_ACTION

ACTION Init_exit:
//write reset state variables to robot.
wr_state(RCts.UR3,RCts.RESET_STATE);
//write reset state variables to robot.
//wr_state(CS.UR5,RESET_STATE);
END_ACTION

ACTION MoveL_active:
//read register from robot and chek is can read 2 or more correct values 
IF ck_state(RCts.UR3,RCts.UR3Move_I) THEN
	 I_STATE:= RCts.UR3Move_I;
ELSIF ck_state(RCts.UR3,RCts.UR3Move_F) THEN
	I_STATE := RCts.UR3Move_F;
END_IF


//read internal variable and write over output variable
Act_In_State := I_STATE;
END_ACTION

ACTION MoveL_entry:
//write state variables to robot, to execute respective state.
wr_state(RCts.UR3,RCts.UR3Move);
//write the retain state variable 
Act_Gl_State:=RCts.UR3Move;
END_ACTION

ACTION MoveL_exit:
//write reset state variables to robot.
wr_state(RCts.UR3,RCts.RESET_STATE);
//reset Global state variable
G_STATE := -1;
END_ACTION

ACTION ReturnR_active:
//read register from robot and chek is can read 2 or more correct values 
IF ck_state(RCts.UR3,RCts.UR3Return_I) THEN
	 I_STATE:= RCts.UR3Return_I;
ELSIF ck_state(RCts.UR3,RCts.UR3Return_F) THEN
	I_STATE := RCts.UR3Return_F;
END_IF

//read internal variable and write over output variable
Act_In_State := I_STATE;
END_ACTION

ACTION ReturnR_entry:
//write state variables to robot, to execute respective state.
wr_state(RCts.UR3,RCts.UR3Return);
//write the retain state variable 
Act_Gl_State:=RCts.UR3Return;
END_ACTION

ACTION ReturnR_exit:
//write reset state variables to robot.
wr_state(RCts.UR3,RCts.RESET_STATE);
//reset Global state variable
G_STATE := -1;
END_ACTION

ACTION UR3Move_entry:
//write state variables to robot, to execute respective state.
wr_state(RCts.UR3,RCts.UR3CatchSeparator);
//write the retain state variable 
Act_Gl_State:=RCts.UR3CatchSeparator;
END_ACTION

ACTION UR3Move_exit:
//write reset state variables to robot.
wr_state(RCts.UR3,RCts.RESET_STATE);
//reset Global state variable
G_STATE := -1;
END_ACTION

ACTION Wrt_FState_entry:
//write output variable to indicate that the robot execute the state 
State_complete := TRUE;
END_ACTION

ACTION Wrt_FState_exit:
//write output variable to indicate that the robot execute the state 
State_complete := FALSE;
//init_:=FALSE;

G_STATE := -1;
//rest internat state variable
I_STATE :=-1;
END_ACTION

END_PROGRAM

// ---- POUs/POUs/ROBOTS/Robot_functions/ck_state.TcPOU
FUNCTION ck_state : BOOL
VAR_INPUT
	robot : INT;
	state : INT;

END_VAR
VAR
	ck0 : INT;
	ck1 : INT;
	ck2 : INT;
END_VAR

//leer del robot al plc
IF robot=3 THEN
ck0 := flip_byte_int(Robot_UR3.UR_outputs_int.INT3);
ck1 := flip_byte_int(Robot_UR3.UR_outputs_int.INT4);
ck2 := flip_byte_int(Robot_UR3.UR_outputs_int.INT5);
ELSIF robot=5 THEN
ck0 := flip_byte_int(Robot_UR5.UR_outputs_int.INT3);
ck1 := flip_byte_int(Robot_UR5.UR_outputs_int.INT4);
ck2 := flip_byte_int(Robot_UR5.UR_outputs_int.INT5);
END_IF

IF (ck0=state AND ck1=state AND ck2=state) OR (ck0<>state AND ck1=state AND ck2=state) OR (ck0=state AND ck1<>state AND ck2=state) OR (ck0=state AND ck1=state AND ck2<>state) THEN
ck_state := TRUE;
ELSE 
ck_state := FALSE;	
END_IF

END_FUNCTION

// ---- POUs/POUs/l/flip_byte_int.TcPOU
FUNCTION flip_byte_int :  INT
VAR_INPUT
	
	byte_array : ARRAY[0..3] OF BYTE;
END_VAR

VAR
		valor_flip : ARRAY[0..3] OF BYTE;
		pt: POINTER TO INT;
		

		
END_VAR


//direcciones


valor_flip[0] := byte_array[3];
valor_flip[1] := byte_array[2];
valor_flip[2] := byte_array[1];
valor_flip[3] := byte_array[0];

pt := ADR(valor_flip);
flip_byte_int := pt^;

END_FUNCTION

// ---- POUs/POUs/ROBOTS/Robot_functions/wr_state.TcPOU
FUNCTION wr_state : BOOL
VAR_INPUT
	function_state : INT;
	state : INT;
END_VAR
VAR
END_VAR

wr_state := FALSE;
//WRITE FLAGS STATE-MACHINE #################(PLC->ROBOT)
//write the UR3 robot integer register to set flag states
IF function_state= RCts.UR3 THEN
Robot_UR3.UR_inputs.Ints.INT0 := flip_int(state);
Robot_UR3.UR_inputs.Ints.INT1 := flip_int(state);
Robot_UR3.UR_inputs.Ints.INT2 := flip_int(state);
wr_state := TRUE;
//write the CS.UR5 robot integer register to set flag states
ELSIF  function_state= RCts.UR5 THEN 
Robot_UR5.UR_inputs.Ints.INT0 := flip_int(state);
Robot_UR5.UR_inputs.Ints.INT1 := flip_int(state);
Robot_UR5.UR_inputs.Ints.INT2 := flip_int(state);
wr_state := TRUE;
END_IF

END_FUNCTION

// ---- POUs/POUs/l/flip_int.TcPOU
FUNCTION flip_int : ARRAY[0..3] OF BYTE
VAR_INPUT
	valor_real : INT;
END_VAR

VAR
		valor_byte :  ARRAY[0..3] OF BYTE;
		valor_flip : ARRAY[0..3] OF BYTE;
		pByteIn1, pByteIn2, pByteIn3, pByteIn4: POINTER TO BYTE;
		

		
END_VAR


//direcciones
pByteIn1 := ADR(valor_real);
pByteIn2 := ADR(valor_real) + SIZEOF(BYTE);
pByteIn3 := ADR(valor_real) + 2 * SIZEOF(BYTE);
pByteIn4 := ADR(valor_real) + 3 * SIZEOF(BYTE);



valor_byte[0] := pByteIn1^;
valor_byte[1] := pByteIn2^ ;
valor_byte[2] := pByteIn3^ ;
valor_byte[3] := pByteIn4^ ;

valor_flip[0] := valor_byte[3];
valor_flip[1] := valor_byte[2];
valor_flip[2] := valor_byte[1];
valor_flip[3] := valor_byte[0];


flip_int := valor_flip;

END_FUNCTION

// ---- POUs/POUs/ROBOTS/Robot_machine_state/UR5_StateMachine.TcPOU
PROGRAM UR5_StateMachine
//FUNCTION_BLOCK
VAR
//internal aux state
I_STATE : INT:=-1;

	//vars to start and stop Robot, safety segurity, power on
	UR5_Safety_pin_1 AT%Q*:BOOL:= FALSE;
	UR5_Safety_pin_2 AT%Q*:BOOL:= FALSE;
	UR5_Power_on AT%Q*:BOOL:= FALSE;
	UR5_Run_Robot AT%Q*:BOOL:= FALSE;


END_VAR


VAR_INPUT
	init_: BOOL:= FALSE;
	G_STATE: INT:=-1;
	Num_Ctr_Cam : INT:=-1;
END_VAR

VAR_OUTPUT
	State_complete : BOOL:= FALSE;
	Act_Gl_State :INT:=-1;
	Act_In_State: INT:=-1;
END_VAR

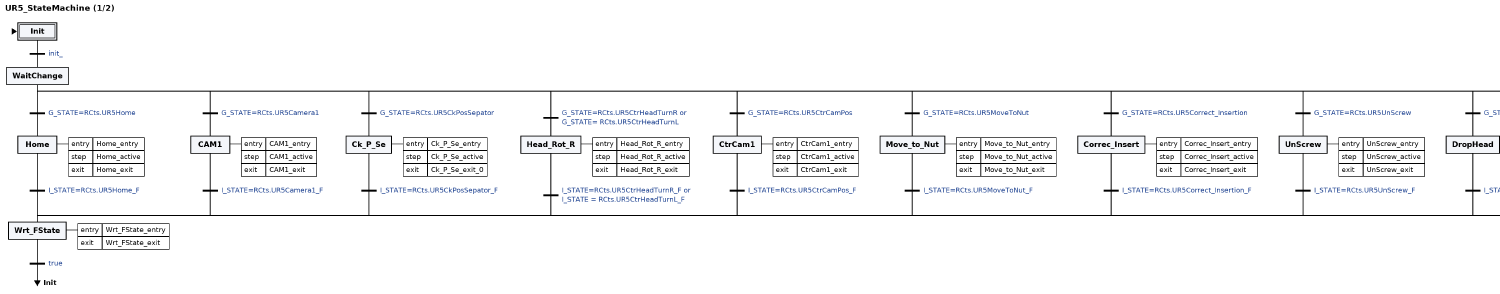
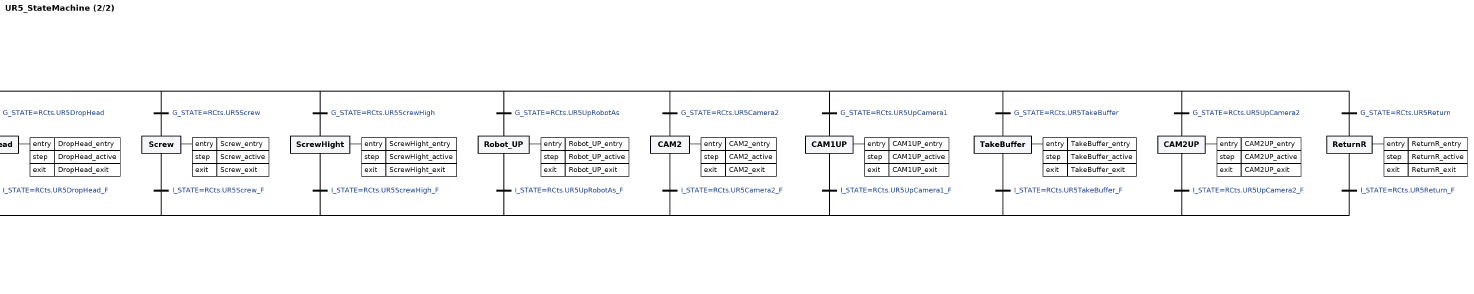
INITIAL_STEP Init:
END_STEP
TRANSITION FROM Init TO WaitChange
    := init_;
END_TRANSITION
STEP WaitChange:
END_STEP
TRANSITION FROM WaitChange TO Home
    := G_STATE=RCts.UR5Home;
END_TRANSITION
STEP Home:
    Home_entry(P1);  // entry action
    Home_active(N);  // step action
    Home_exit(P0);  // exit action
END_STEP
TRANSITION FROM Home TO Wrt_FState
    := I_STATE=RCts.UR5Home_F;
END_TRANSITION
TRANSITION FROM WaitChange TO CAM1
    := G_STATE=RCts.UR5Camera1;
END_TRANSITION
STEP CAM1:
    CAM1_entry(P1);  // entry action
    CAM1_active(N);  // step action
    CAM1_exit(P0);  // exit action
END_STEP
TRANSITION FROM CAM1 TO Wrt_FState
    := I_STATE=RCts.UR5Camera1_F;
END_TRANSITION
TRANSITION FROM WaitChange TO Ck_P_Se
    := G_STATE=RCts.UR5CkPosSepator;
END_TRANSITION
STEP Ck_P_Se:
    Ck_P_Se_entry(P1);  // entry action
    Ck_P_Se_active(N);  // step action
    Ck_P_Se_exit_0(P0);  // exit action
END_STEP
TRANSITION FROM Ck_P_Se TO Wrt_FState
    := I_STATE=RCts.UR5CkPosSepator_F;
END_TRANSITION
TRANSITION FROM WaitChange TO Head_Rot_R
    := G_STATE=RCts.UR5CtrHeadTurnR or G_STATE= RCts.UR5CtrHeadTurnL;
END_TRANSITION
STEP Head_Rot_R:
    Head_Rot_R_entry(P1);  // entry action
    Head_Rot_R_active(N);  // step action
    Head_Rot_R_exit(P0);  // exit action
END_STEP
TRANSITION FROM Head_Rot_R TO Wrt_FState
    := I_STATE=RCts.UR5CtrHeadTurnR_F or I_STATE = RCts.UR5CtrHeadTurnL_F;
END_TRANSITION
TRANSITION FROM WaitChange TO CtrCam1
    := G_STATE=RCts.UR5CtrCamPos;
END_TRANSITION
STEP CtrCam1:
    CtrCam1_entry(P1);  // entry action
    CtrCam1_active(N);  // step action
    CtrCam1_exit(P0);  // exit action
END_STEP
TRANSITION FROM CtrCam1 TO Wrt_FState
    := I_STATE=RCts.UR5CtrCamPos_F;
END_TRANSITION
TRANSITION FROM WaitChange TO Move_to_Nut
    := G_STATE=RCts.UR5MoveToNut;
END_TRANSITION
STEP Move_to_Nut:
    Move_to_Nut_entry(P1);  // entry action
    Move_to_Nut_active(N);  // step action
    Move_to_Nut_exit(P0);  // exit action
END_STEP
TRANSITION FROM Move_to_Nut TO Wrt_FState
    := I_STATE=RCts.UR5MoveToNut_F;
END_TRANSITION
TRANSITION FROM WaitChange TO Correc_Insert
    := G_STATE=RCts.UR5Correct_Insertion;
END_TRANSITION
STEP Correc_Insert:
    Correc_Insert_entry(P1);  // entry action
    Correc_Insert_active(N);  // step action
    Correc_Insert_exit(P0);  // exit action
END_STEP
TRANSITION FROM Correc_Insert TO Wrt_FState
    := I_STATE=RCts.UR5Correct_Insertion_F;
END_TRANSITION
TRANSITION FROM WaitChange TO UnScrew
    := G_STATE=RCts.UR5UnScrew;
END_TRANSITION
STEP UnScrew:
    UnScrew_entry(P1);  // entry action
    UnScrew_active(N);  // step action
    UnScrew_exit(P0);  // exit action
END_STEP
TRANSITION FROM UnScrew TO Wrt_FState
    := I_STATE=RCts.UR5UnScrew_F;
END_TRANSITION
TRANSITION FROM WaitChange TO DropHead
    := G_STATE=RCts.UR5DropHead;
END_TRANSITION
STEP DropHead:
    DropHead_entry(P1);  // entry action
    DropHead_active(N);  // step action
    DropHead_exit(P0);  // exit action
END_STEP
TRANSITION FROM DropHead TO Wrt_FState
    := I_STATE=RCts.UR5DropHead_F;
END_TRANSITION
TRANSITION FROM WaitChange TO Screw
    := G_STATE=RCts.UR5Screw;
END_TRANSITION
STEP Screw:
    Screw_entry(P1);  // entry action
    Screw_active(N);  // step action
    Screw_exit(P0);  // exit action
END_STEP
TRANSITION FROM Screw TO Wrt_FState
    := I_STATE=RCts.UR5Screw_F;
END_TRANSITION
TRANSITION FROM WaitChange TO ScrewHight
    := G_STATE=RCts.UR5ScrewHigh;
END_TRANSITION
STEP ScrewHight:
    ScrewHight_entry(P1);  // entry action
    ScrewHight_active(N);  // step action
    ScrewHight_exit(P0);  // exit action
END_STEP
TRANSITION FROM ScrewHight TO Wrt_FState
    := I_STATE=RCts.UR5ScrewHigh_F;
END_TRANSITION
TRANSITION FROM WaitChange TO Robot_UP
    := G_STATE=RCts.UR5UpRobotAs;
END_TRANSITION
STEP Robot_UP:
    Robot_UP_entry(P1);  // entry action
    Robot_UP_active(N);  // step action
    Robot_UP_exit(P0);  // exit action
END_STEP
TRANSITION FROM Robot_UP TO Wrt_FState
    := I_STATE=RCts.UR5UpRobotAs_F;
END_TRANSITION
TRANSITION FROM WaitChange TO CAM2
    := G_STATE=RCts.UR5Camera2;
END_TRANSITION
STEP CAM2:
    CAM2_entry(P1);  // entry action
    CAM2_active(N);  // step action
    CAM2_exit(P0);  // exit action
END_STEP
TRANSITION FROM CAM2 TO Wrt_FState
    := I_STATE=RCts.UR5Camera2_F;
END_TRANSITION
TRANSITION FROM WaitChange TO CAM1UP
    := G_STATE=RCts.UR5UpCamera1;
END_TRANSITION
STEP CAM1UP:
    CAM1UP_entry(P1);  // entry action
    CAM1UP_active(N);  // step action
    CAM1UP_exit(P0);  // exit action
END_STEP
TRANSITION FROM CAM1UP TO Wrt_FState
    := I_STATE=RCts.UR5UpCamera1_F;
END_TRANSITION
TRANSITION FROM WaitChange TO TakeBuffer
    := G_STATE=RCts.UR5TakeBuffer;
END_TRANSITION
STEP TakeBuffer:
    TakeBuffer_entry(P1);  // entry action
    TakeBuffer_active(N);  // step action
    TakeBuffer_exit(P0);  // exit action
END_STEP
TRANSITION FROM TakeBuffer TO Wrt_FState
    := I_STATE=RCts.UR5TakeBuffer_F;
END_TRANSITION
TRANSITION FROM WaitChange TO CAM2UP
    := G_STATE=RCts.UR5UpCamera2;
END_TRANSITION
STEP CAM2UP:
    CAM2UP_entry(P1);  // entry action
    CAM2UP_active(N);  // step action
    CAM2UP_exit(P0);  // exit action
END_STEP
TRANSITION FROM CAM2UP TO Wrt_FState
    := I_STATE=RCts.UR5UpCamera2_F;
END_TRANSITION
TRANSITION FROM WaitChange TO ReturnR
    := G_STATE=RCts.UR5Return;
END_TRANSITION
STEP ReturnR:
    ReturnR_entry(P1);  // entry action
    ReturnR_active(N);  // step action
    ReturnR_exit(P0);  // exit action
END_STEP
TRANSITION FROM ReturnR TO Wrt_FState
    := I_STATE=RCts.UR5Return_F;
END_TRANSITION
STEP Wrt_FState:
    Wrt_FState_entry(P1);  // entry action
    Wrt_FState_exit(P0);  // exit action
END_STEP
TRANSITION FROM Wrt_FState TO Init
    := true;
END_TRANSITION

ACTION CAM1_active:
//read register from robot and chek is can read 2 or more correct values 
IF ck_state(RCts.UR5,RCts.UR5Camera1_I) THEN
	 I_STATE:= RCts.UR5Camera1_I;
ELSIF ck_state(RCts.UR5,RCts.UR5Camera1_F) THEN
	I_STATE := RCts.UR5Camera1_F;
END_IF

//read internal variable and write over output variable
Act_In_State := I_STATE;
END_ACTION

ACTION CAM1_entry:
//write state variables to robot, to execute respective state.
wr_state(RCts.UR5,RCts.UR5Camera1);
//write the retain state variable 
Act_Gl_State:=RCts.UR5Camera1;
END_ACTION

ACTION CAM1_exit:
//write reset state variables to robot.
wr_state(RCts.UR5,RCts.RESET_STATE);
//reset Global state variable
G_STATE := -1;
END_ACTION

ACTION CAM1UP_active:
//read register from robot and chek is can read 2 or more correct values 
IF ck_state(RCts.UR5,RCts.UR5UpCamera1_I) THEN
	 I_STATE:= RCts.UR5UpCamera1_I;
ELSIF ck_state(RCts.UR5,RCts.UR5UpCamera1_F) THEN
	I_STATE := RCts.UR5UpCamera1_F;
END_IF

//read internal variable and write over output variable
Act_In_State := I_STATE;
END_ACTION

ACTION CAM1UP_entry:
//write state variables to robot, to execute respective state.
wr_state(RCts.UR5,RCts.UR5UpCamera1);
//write the retain state variable 
Act_Gl_State:=RCts.UR5UpCamera1;
END_ACTION

ACTION CAM1UP_exit:
//write reset state variables to robot.
wr_state(RCts.UR5,RCts.RESET_STATE);
//reset Global state variable
G_STATE := -1;
END_ACTION

ACTION CAM2_active:
//read register from robot and chek is can read 2 or more correct values 
IF ck_state(RCts.UR5,RCts.UR5Camera2_I) THEN
	 I_STATE:= RCts.UR5Camera2_I;
ELSIF ck_state(RCts.UR5,RCts.UR5Camera2_F) THEN
	I_STATE := RCts.UR5Camera2_F;
END_IF



//read internal variable and write over output variable
Act_In_State := I_STATE;
END_ACTION

ACTION CAM2_entry:
//write state variables to robot, to execute respective state.
wr_state(RCts.UR5,RCts.UR5Camera2);
//write the retain state variable 
Act_Gl_State:=RCts.UR5Camera2;
END_ACTION

ACTION CAM2_exit:

//write reset state variables to robot.
wr_state(RCts.UR5,RCts.RESET_STATE);
//reset Global state variable
G_STATE := -1;
END_ACTION

ACTION CAM2UP_active:
//read register from robot and chek is can read 2 or more correct values 
IF ck_state(RCts.UR5,RCts.UR5UpCamera2_I) THEN
	 I_STATE:= RCts.UR5UpCamera2_I;
ELSIF ck_state(RCts.UR5,RCts.UR5UpCamera2_F) THEN
	I_STATE := RCts.UR5UpCamera2_F;
END_IF


//read internal variable and write over output variable
Act_In_State := I_STATE;
END_ACTION

ACTION CAM2UP_entry:
//write state variables to robot, to execute respective state.
wr_state(RCts.UR5,RCts.UR5UpCamera2);
//write the retain state variable 
Act_Gl_State:=RCts.UR5UpCamera2;
END_ACTION

ACTION CAM2UP_exit:
//write reset state variables to robot.
wr_state(RCts.UR5,RCts.RESET_STATE);
//reset Global state variable
G_STATE := -1;
END_ACTION

ACTION Ck_P_Se_active:
//read register from robot and chek is can read 2 or more correct values 
IF ck_state(RCts.UR5,RCts.UR5CkPosSepator_I) THEN
	 I_STATE:= RCts.UR5CkPosSepator_I;
ELSIF ck_state(RCts.UR5,RCts.UR5CkPosSepator_F) THEN
	I_STATE := RCts.UR5CkPosSepator_F;
END_IF


//read internal variable and write over output variable
Act_In_State := I_STATE;
END_ACTION

ACTION Ck_P_Se_entry:
//write state variables to robot, to execute respective state.
wr_state(RCts.UR5,RCts.UR5CkPosSepator);
//write the retain state variable 
Act_Gl_State:=RCts.UR5CkPosSepator;
END_ACTION

ACTION Ck_P_Se_exit:
// NETWORK 1
END_ACTION

ACTION Ck_P_Se_exit_0:
//write reset state variables to robot.
wr_state(RCts.UR5,RCts.RESET_STATE);
//reset Global state variable
G_STATE := -1;
I_STATE := -1;
END_ACTION

ACTION Correc_Insert_active:


//send normal force UR3->Ur5
wr_real_value(RCts.UR_DATA_SEND,flip_byte(Robot_UR3.UR_TCP.FLOAT14));
//read register from robot and chek is can read 2 or more correct values 
IF ck_state(RCts.UR5,RCts.UR5Correct_Insertion_I) THEN
	 I_STATE:= RCts.UR5Correct_Insertion_I;
ELSIF ck_state(RCts.UR5,RCts.UR5Correct_Insertion_F) THEN
	I_STATE := RCts.UR5Correct_Insertion_F;
END_IF

//

//read internal variable and write over output variable
Act_In_State := I_STATE;
END_ACTION

ACTION Correc_Insert_entry:
//write state variables to robot, to execute respective state.
wr_state(RCts.UR5,RCts.UR5Correct_Insertion);
//write the retain state variable 
Act_Gl_State:=RCts.UR5Correct_Insertion;
END_ACTION

ACTION Correc_Insert_exit:
//write reset state variables to robot.
wr_state(RCts.UR5,RCts.RESET_STATE);
//reset Global state variable
G_STATE := -1;
END_ACTION

ACTION CtrCam1_active:

//read register from robot and chek is can read 2 or more correct values 
IF ck_state(RCts.UR5,RCts.UR5CtrCamPos_I) THEN
	 I_STATE:= RCts.UR5CtrCamPos_I;
ELSIF ck_state(RCts.UR5,RCts.UR5CtrCamPos_F) THEN
	I_STATE := RCts.UR5CtrCamPos_F;
END_IF


//read internal variable and write over output variable
Act_In_State := I_STATE;
END_ACTION

ACTION CtrCam1_entry:


CASE Num_Ctr_Cam OF 
	1:
		//write state variables to robot, to execute respective state.
		wr_state(RCts.UR5,RCts.UR5CtrCamPos1);
		//write the retain state variable 
		Act_Gl_State:=RCts.UR5CtrCamPos1;
	2:
		//write state variables to robot, to execute respective state.
		wr_state(RCts.UR5,RCts.UR5CtrCamPos2);
		//write the retain state variable 
		Act_Gl_State:=RCts.UR5CtrCamPos2;
	3:
		//write state variables to robot, to execute respective state.
		wr_state(RCts.UR5,RCts.UR5CtrCamPos3);
		//write the retain state variable 
		Act_Gl_State:=RCts.UR5CtrCamPos3;
	4:
		//write state variables to robot, to execute respective state.
		wr_state(RCts.UR5,RCts.UR5CtrCamPos4);
		//write the retain state variable 
		Act_Gl_State:=RCts.UR5CtrCamPos4;
	
END_CASE
END_ACTION

ACTION CtrCam1_exit:
//write reset state variables to robot.
wr_state(RCts.UR5,RCts.RESET_STATE);
//reset Global state variable
G_STATE := -1;
END_ACTION

ACTION DropHead_active:
//read register from robot and chek is can read 2 or more correct values 
IF ck_state(RCts.UR5,RCts.UR5DropHead_I) THEN
	 I_STATE:= RCts.UR5DropHead_I;
ELSIF ck_state(RCts.UR5,RCts.UR5DropHead_F) THEN
	I_STATE := RCts.UR5DropHead_F;
END_IF



//read internal variable and write over output variable
Act_In_State := I_STATE;
END_ACTION

ACTION DropHead_entry:
//write state variables to robot, to execute respective state.
wr_state(RCts.UR5,RCts.UR5DropHead);
//write the retain state variable 
Act_Gl_State:=RCts.UR5DropHead;
END_ACTION

ACTION DropHead_exit:

//write reset state variables to robot.
wr_state(RCts.UR5,RCts.RESET_STATE);
//reset Global state variable
G_STATE := -1;
END_ACTION

ACTION Head_Rot_R_active:


IF Num_Ctr_Cam = 1 THEN
	//read register from robot and chek is can read 2 or more correct values 
	IF ck_state(RCts.UR5,RCts.UR5CtrHeadTurnR_I) THEN
		 I_STATE:= RCts.UR5CtrHeadTurnR_I;
	ELSIF ck_state(RCts.UR5,RCts.UR5CtrHeadTurnR_F) THEN
		I_STATE := RCts.UR5CtrHeadTurnR_F;
	END_IF

ELSIF Num_Ctr_Cam = 2 THEN 
		//read register from robot and chek is can read 2 or more correct values 
	IF ck_state(RCts.UR5,RCts.UR5CtrHeadTurnL_I) THEN
		 I_STATE:= RCts.UR5CtrHeadTurnR_I;
	ELSIF ck_state(RCts.UR5,RCts.UR5CtrHeadTurnL_F) THEN
		I_STATE := RCts.UR5CtrHeadTurnL_F;
	END_IF

END_IF




//read internal variable and write over output variable
Act_In_State := I_STATE;
END_ACTION

ACTION Head_Rot_R_entry:
//write state variables to robot, to execute respective state.

IF Num_Ctr_Cam = 1 THEN
	wr_state(RCts.UR5,RCts.UR5CtrHeadTurnR);
	//write the retain state variable 
	Act_Gl_State:=RCts.UR5CtrHeadTurnR;
ELSIF Num_Ctr_Cam = 2 THEN 
	wr_state(RCts.UR5,RCts.UR5CtrHeadTurnL);
	//write the retain state variable 
	Act_Gl_State:=RCts.UR5CtrHeadTurnL;	
END_IF
END_ACTION

ACTION Head_Rot_R_exit:
//write reset state variables to robot.
wr_state(RCts.UR5,RCts.RESET_STATE);
//reset Global state variable
G_STATE := -1;
I_STATE := -1;
END_ACTION

ACTION Home_active:
//read register from robot and chek is can read 2 or more correct values 
IF ck_state(RCts.UR5,RCts.UR5Home_I) THEN
	 I_STATE:= RCts.UR5Home_I;
ELSIF ck_state(RCts.UR5,RCts.UR5Home_F) THEN
	I_STATE := RCts.UR5Home_F;
END_IF


//read internal variable and write over output variable
Act_In_State := I_STATE;
END_ACTION

ACTION Home_entry:
//write state variables to robot, to execute respective state.
wr_state(RCts.UR5,RCts.UR5Home);
//write the retain state variable 
Act_Gl_State:=RCts.UR5Home;
END_ACTION

ACTION Home_exit:
//write reset state variables to robot.
wr_state(RCts.UR5,RCts.RESET_STATE);
//reset Global state variable
G_STATE := -1;
END_ACTION

ACTION Move_robot_active:
//read register from robot and chek is can read 2 or more correct values 
IF ck_state(RCts.UR5,RCts.UR5CkPosSepator_I) THEN
	 I_STATE:= RCts.UR5CkPosSepator_I;
ELSIF ck_state(RCts.UR5,RCts.UR5CkPosSepator_F) THEN
	I_STATE := RCts.UR5CkPosSepator_F;
END_IF
END_ACTION

ACTION Move_robot_entry:
//get the value of neural network and save
//SepPositions[aux_cnt_SepPos] := Vision_struct.Pos_sep.Val1;
//aux_cnt_SepPos := aux_cnt_SepPos + 1;

//set the Robot_vision Flags to indicate vision system finish (PLC->Robot)
write_bool_flag(TRUE);
END_ACTION

ACTION Move_to_Nut_active:
//send normal force UR3->Ur5
//float 18 norm force 
//
wr_real_value(RCts.UR_DATA_SEND,flip_byte(Robot_UR3.UR_TCP.FLOAT14));

//read register from robot and chek is can read 2 or more correct values 
IF ck_state(RCts.UR5,RCts.UR5MoveToNut_I) THEN
	 I_STATE:= RCts.UR5MoveToNut_I;
ELSIF ck_state(RCts.UR5,RCts.UR5MoveToNut_F) THEN
	I_STATE := RCts.UR5MoveToNut_F;
END_IF


//read internal variable and write over output variable
Act_In_State := I_STATE;
END_ACTION

ACTION Move_to_Nut_entry:

CASE Num_Ctr_Cam OF 
	1:
		//write state variables to robot, to execute respective state.
		wr_state(RCts.UR5,RCts.UR5MoveToNut1);
		//write the retain state variable 
		Act_Gl_State:=RCts.UR5MoveToNut1;
	2:
		//write state variables to robot, to execute respective state.
		wr_state(RCts.UR5,RCts.UR5MoveToNut2);
		//write the retain state variable 
		Act_Gl_State:=RCts.UR5MoveToNut2;
	3:
		//write state variables to robot, to execute respective state.
		wr_state(RCts.UR5,RCts.UR5MoveToNut3);
		//write the retain state variable 
		Act_Gl_State:=RCts.UR5MoveToNut3;
	4:
		//write state variables to robot, to execute respective state.
		wr_state(RCts.UR5,RCts.UR5MoveToNut4);
		//write the retain state variable 
		Act_Gl_State:=RCts.UR5MoveToNut4;
	
END_CASE
END_ACTION

ACTION Move_to_Nut_exit:

//write reset state variables to robot.
wr_state(RCts.UR5,RCts.RESET_STATE);
//reset Global state variable
G_STATE := -1;
END_ACTION

ACTION ReturnR_active:
//read register from robot and chek is can read 2 or more correct values 
IF ck_state(RCts.UR5,RCts.UR5Return_I) THEN
	 I_STATE:= RCts.UR5Return_I;
ELSIF ck_state(RCts.UR5,RCts.UR5Return_F) THEN
	I_STATE := RCts.UR5Return_F;
END_IF


//read internal variable and write over output variable
Act_In_State := I_STATE;
END_ACTION

ACTION ReturnR_entry:
//write state variables to robot, to execute respective state.
wr_state(RCts.UR5,RCts.UR5Return);
//write the retain state variable 
Act_Gl_State:=RCts.UR5Return;
END_ACTION

ACTION ReturnR_exit:
//write reset state variables to robot.
wr_state(RCts.UR5,RCts.RESET_STATE);
//reset Global state variable
G_STATE := -1;
END_ACTION

ACTION Robot_UP_active:


//read register from robot and chek is can read 2 or more correct values 
IF ck_state(RCts.UR5,RCts.UR5UpRobotAs_I) THEN
	 I_STATE:= RCts.UR5UpRobotAs_I;
ELSIF ck_state(RCts.UR5,RCts.UR5UpRobotAs_F) THEN
	I_STATE := RCts.UR5UpRobotAs_F;
END_IF

//

//read internal variable and write over output variable
Act_In_State := I_STATE;
END_ACTION

ACTION Robot_UP_entry:
//write state variables to robot, to execute respective state.
wr_state(RCts.UR5,RCts.UR5UpRobotAs);
//write the retain state variable 
Act_Gl_State:=RCts.UR5UpRobotAs;
END_ACTION

ACTION Robot_UP_exit:
//write reset state variables to robot.
wr_state(RCts.UR5,RCts.RESET_STATE);
//reset Global state variable
G_STATE := -1;
END_ACTION

ACTION Screw_active:
//read register from robot and chek is can read 2 or more correct values 
IF ck_state(RCts.UR5,RCts.UR5Screw_I) THEN
	 I_STATE:= RCts.UR5Screw_I;
ELSIF ck_state(RCts.UR5,RCts.UR5Screw_F) THEN
	I_STATE := RCts.UR5Screw_F;
END_IF

//

//read internal variable and write over output variable
Act_In_State := I_STATE;
END_ACTION

ACTION Screw_entry:
//write state variables to robot, to execute respective state.
wr_state(RCts.UR5,RCts.UR5Screw);
//write the retain state variable 
Act_Gl_State:=RCts.UR5Screw;
END_ACTION

ACTION Screw_exit:
//write reset state variables to robot.
wr_state(RCts.UR5,RCts.RESET_STATE);
//reset Global state variable
G_STATE := -1;
END_ACTION

ACTION ScrewHight_active:
//read register from robot and chek is can read 2 or more correct values 
IF ck_state(RCts.UR5,RCts.UR5ScrewHigh_I) THEN
	 I_STATE:= RCts.UR5ScrewHigh_I;
ELSIF ck_state(RCts.UR5,RCts.UR5ScrewHigh_F) THEN
	I_STATE := RCts.UR5ScrewHigh_F;
END_IF

//

//read internal variable and write over output variable
Act_In_State := I_STATE;
END_ACTION

ACTION ScrewHight_entry:
//write state variables to robot, to execute respective state.
wr_state(RCts.UR5,RCts.UR5ScrewHigh);
//write the retain state variable 
Act_Gl_State:=RCts.UR5ScrewHigh;
END_ACTION

ACTION ScrewHight_exit:
//write reset state variables to robot.
wr_state(RCts.UR5,RCts.RESET_STATE);
//reset Global state variable
G_STATE := -1;
END_ACTION

ACTION TakeBuffer_active:
//read register from robot and chek is can read 2 or more correct values 
IF ck_state(RCts.UR5,RCts.UR5TakeBuffer_I) THEN
	 I_STATE:= RCts.UR5TakeBuffer_I;
ELSIF ck_state(RCts.UR5,RCts.UR5TakeBuffer_F) THEN
	I_STATE := RCts.UR5TakeBuffer_F;
END_IF

//read internal variable and write over output variable
Act_In_State := I_STATE;
END_ACTION

ACTION TakeBuffer_entry:
//write state variables to robot, to execute respective state.
wr_state(RCts.UR5,RCts.UR5TakeBuffer);
//write the retain state variable 
Act_Gl_State:=RCts.UR5TakeBuffer;
END_ACTION

ACTION TakeBuffer_exit:
//write reset state variables to robot.
wr_state(RCts.UR5,RCts.RESET_STATE);
//reset Global state variable
G_STATE := -1;
I_STATE := -1;
END_ACTION

ACTION UnScrew_active:
//read register from robot and chek is can read 2 or more correct values 
IF ck_state(RCts.UR5,RCts.UR5UnScrew_I) THEN
	 I_STATE:= RCts.UR5UnScrew_I;
ELSIF ck_state(RCts.UR5,RCts.UR5UnScrew_F) THEN
	I_STATE := RCts.UR5UnScrew_F;
END_IF

//

//read internal variable and write over output variable
Act_In_State := I_STATE;
END_ACTION

ACTION UnScrew_entry:
//write state variables to robot, to execute respective state.
wr_state(RCts.UR5,RCts.UR5UnScrew);
//write the retain state variable 
Act_Gl_State:=RCts.UR5UnScrew;
END_ACTION

ACTION UnScrew_exit:
//write reset state variables to robot.
wr_state(RCts.UR5,RCts.RESET_STATE);
//reset Global state variable
G_STATE := -1;
END_ACTION

ACTION Wrt_FState_entry:
//write output variable to indicate that the robot execute the state 
State_complete := TRUE;
END_ACTION

ACTION Wrt_FState_exit:
//write output variable to indicate that the robot execute the state 
State_complete := FALSE;
END_ACTION

END_PROGRAM

// ---- POUs/POUs/VISION/Vision_functions/wr_real_value.TcPOU
FUNCTION wr_real_value : BOOL
VAR_INPUT
	function_state : INT;
	value : REAL;
END_VAR
VAR
END_VAR

wr_real_value := FALSE;

//#####################	WRITE VISION VARIABLES #################(PLC->ROBOT)
//write the CS.UR5 robot float register to send CX position
IF  function_state= VCts.CX_VALUE THEN
Robot_UR5.UR_inputs.Floats.FLOAT0 := flip_real(value);
Robot_UR5.UR_inputs.Floats.FLOAT1 := flip_real(value);
Robot_UR5.UR_inputs.Floats.FLOAT2 := flip_real(value);
wr_real_value := TRUE;
//write the CS.UR5 robot float register to send CY position
ELSIF  function_state= VCts.CY_VALUE THEN
Robot_UR5.UR_inputs.Floats.FLOAT3 := flip_real(value);
Robot_UR5.UR_inputs.Floats.FLOAT4 := flip_real(value);
Robot_UR5.UR_inputs.Floats.FLOAT5 := flip_real(value);
wr_real_value := TRUE;
//write the CS.UR5 robot float register to send NUT_TURN position
ELSIF  function_state= VCts.NUT_VALUE THEN
Robot_UR5.UR_inputs.Floats.FLOAT6 := flip_real(value);
Robot_UR5.UR_inputs.Floats.FLOAT7 := flip_real(value);
Robot_UR5.UR_inputs.Floats.FLOAT8 := flip_real(value);
wr_real_value := TRUE;
//write the CS.UR5 robot float register to send HEAD_RIGTH_VALUE position
ELSIF  function_state= VCts.HEAD_RIGTH_VALUE THEN
Robot_UR5.UR_inputs.Floats.FLOAT9 := flip_real(value);
Robot_UR5.UR_inputs.Floats.FLOAT10 := flip_real(value);
Robot_UR5.UR_inputs.Floats.FLOAT11 := flip_real(value);
wr_real_value := TRUE;
//write the CS.UR5 robot float register to send HEAD_LEFT_VALUE position
ELSIF  function_state = VCts.HEAD_LEFT_VALUE THEN
Robot_UR5.UR_inputs_2.Floats.FLOAT12 := flip_real(value);
Robot_UR5.UR_inputs_2.Floats.FLOAT13 := flip_real(value);
Robot_UR5.UR_inputs_2.Floats.FLOAT14:= flip_real(value);
wr_real_value := TRUE;
//write the CS.UR5 robot float register to send NUT_POS_VALUE position
ELSIF  function_state = VCts.SEP_POS_VALUE THEN
Robot_UR5.UR_inputs_2.Floats.FLOAT12 := flip_real(value);
Robot_UR5.UR_inputs_2.Floats.FLOAT13 := flip_real(value);
Robot_UR5.UR_inputs_2.Floats.FLOAT14:= flip_real(value);
wr_real_value := TRUE;
ELSIF  function_state = Rcts.UR_DATA_SEND THEN
Robot_UR5.UR_inputs_2.Floats.FLOAT15 := flip_real(value);
Robot_UR5.UR_inputs_2.Floats.FLOAT16 := flip_real(value);
Robot_UR5.UR_inputs_2.Floats.FLOAT17:= flip_real(value);
wr_real_value := TRUE;
END_IF
wr_real_value := FALSE;

END_FUNCTION

// ---- POUs/POUs/l/flip_real.TcPOU
FUNCTION flip_real : ARRAY[0..3] OF BYTE
VAR_INPUT
	valor_real : REAL;
END_VAR

VAR
		valor_byte :  ARRAY[0..3] OF BYTE;
		valor_flip : ARRAY[0..3] OF BYTE;
		pByteIn1, pByteIn2, pByteIn3, pByteIn4: POINTER TO BYTE;
		

		
END_VAR


//direcciones
pByteIn1 := ADR(valor_real);
pByteIn2 := ADR(valor_real) + SIZEOF(BYTE);
pByteIn3 := ADR(valor_real) + 2 * SIZEOF(BYTE);
pByteIn4 := ADR(valor_real) + 3 * SIZEOF(BYTE);



valor_byte[0] := pByteIn1^;
valor_byte[1] := pByteIn2^ ;
valor_byte[2] := pByteIn3^ ;
valor_byte[3] := pByteIn4^ ;

valor_flip[0] := valor_byte[3];
valor_flip[1] := valor_byte[2];
valor_flip[2] := valor_byte[1];
valor_flip[3] := valor_byte[0];


flip_real := valor_flip;

END_FUNCTION

// ---- POUs/POUs/l/flip_byte.TcPOU
FUNCTION flip_byte :  REAL
VAR_INPUT
	
	byte_array : ARRAY[0..3] OF BYTE;
END_VAR

VAR
		valor_flip : ARRAY[0..3] OF BYTE;
		pt: POINTER TO REAL;
		

		
END_VAR


//direcciones


valor_flip[0] := byte_array[3];
valor_flip[1] := byte_array[2];
valor_flip[2] := byte_array[1];
valor_flip[3] := byte_array[0];

pt := ADR(valor_flip);
flip_byte := pt^;

END_FUNCTION

// ---- POUs/POUs/ROBOTS/Robot_functions/write_bool_flag.TcPOU
FUNCTION write_bool_flag : BOOL
VAR_INPUT
	value : BOOL;
END_VAR
VAR
END_VAR

//Write bit register from PLC to Robot
//Flag to send to robot and indicate when the  system finish its process

write_bool_flag := FALSE;
Robot_UR5.UR_inputs.Bits.B0 := value;
Robot_UR5.UR_inputs.Bits.B1 := value;
Robot_UR5.UR_inputs.Bits.B2 := value;
write_bool_flag := TRUE;

END_FUNCTION

// ---- POUs/POUs/VISION/Vision_machines_states/Vision_StateMachine.TcPOU
PROGRAM  Vision_StateMachine
//PROGRAM Vision_StateMachine
VAR
//var to get struct data from ck_real_value function
cx_vision_data : ck_real_flag_data;
cy_vision_data : ck_real_flag_data;
nut_turn_data : ck_real_flag_data;

sep_pos_data : ck_real_flag_data;

sep_rot_rigth_data :ck_real_flag_data;
sep_rot_left_data :ck_real_flag_data;


//internal aux state
I_STATE : INT:=-1;
	Val1: INT;
END_VAR

VAR_INPUT
init_: BOOL:= FALSE;
//global aux state
G_STATE: INT:=-1;

Aux_State_val :INT := -1;

END_VAR


VAR_OUTPUT
	State_complete : BOOL:= FALSE;
	Act_Gl_State :INT:=-1;
	Act_In_State: INT:=-1;
END_VAR

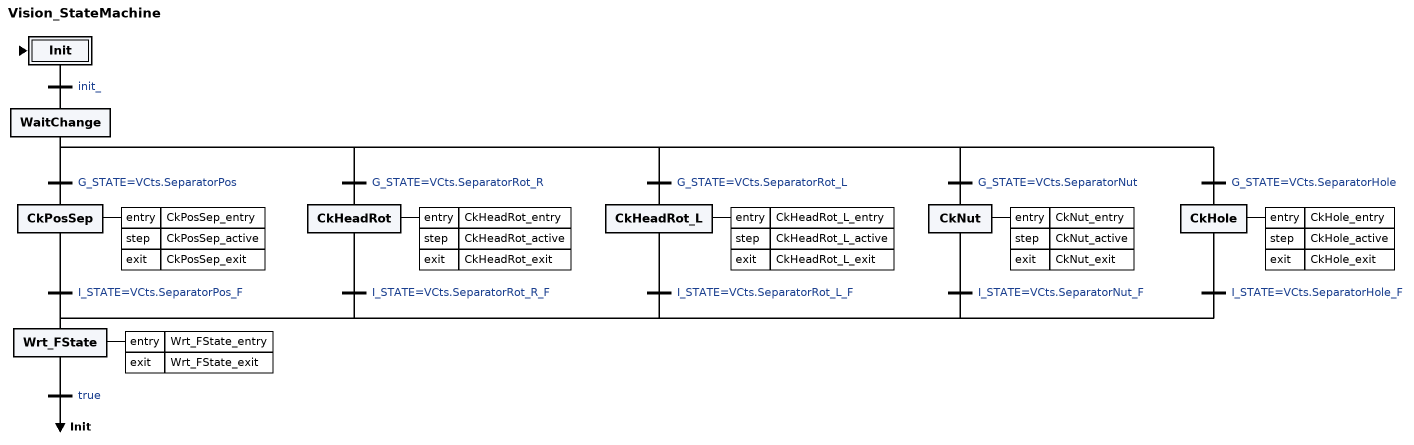
INITIAL_STEP Init:
END_STEP
TRANSITION FROM Init TO WaitChange
    := init_;
END_TRANSITION
STEP WaitChange:
END_STEP
TRANSITION FROM WaitChange TO CkPosSep
    := G_STATE=VCts.SeparatorPos;
END_TRANSITION
STEP CkPosSep:
    CkPosSep_entry(P1);  // entry action
    CkPosSep_active(N);  // step action
    CkPosSep_exit(P0);  // exit action
END_STEP
TRANSITION FROM CkPosSep TO Wrt_FState
    := I_STATE=VCts.SeparatorPos_F;
END_TRANSITION
TRANSITION FROM WaitChange TO CkHeadRot
    := G_STATE=VCts.SeparatorRot_R;
END_TRANSITION
STEP CkHeadRot:
    CkHeadRot_entry(P1);  // entry action
    CkHeadRot_active(N);  // step action
    CkHeadRot_exit(P0);  // exit action
END_STEP
TRANSITION FROM CkHeadRot TO Wrt_FState
    := I_STATE=VCts.SeparatorRot_R_F;
END_TRANSITION
TRANSITION FROM WaitChange TO CkHeadRot_L
    := G_STATE=VCts.SeparatorRot_L;
END_TRANSITION
STEP CkHeadRot_L:
    CkHeadRot_L_entry(P1);  // entry action
    CkHeadRot_L_active(N);  // step action
    CkHeadRot_L_exit(P0);  // exit action
END_STEP
TRANSITION FROM CkHeadRot_L TO Wrt_FState
    := I_STATE=VCts.SeparatorRot_L_F;
END_TRANSITION
TRANSITION FROM WaitChange TO CkNut
    := G_STATE=VCts.SeparatorNut;
END_TRANSITION
STEP CkNut:
    CkNut_entry(P1);  // entry action
    CkNut_active(N);  // step action
    CkNut_exit(P0);  // exit action
END_STEP
TRANSITION FROM CkNut TO Wrt_FState
    := I_STATE=VCts.SeparatorNut_F;
END_TRANSITION
TRANSITION FROM WaitChange TO CkHole
    := G_STATE=VCts.SeparatorHole;
END_TRANSITION
STEP CkHole:
    CkHole_entry(P1);  // entry action
    CkHole_active(N);  // step action
    CkHole_exit(P0);  // exit action
END_STEP
TRANSITION FROM CkHole TO Wrt_FState
    := I_STATE=VCts.SeparatorHole_F;
END_TRANSITION
STEP Wrt_FState:
    Wrt_FState_entry(P1);  // entry action
    Wrt_FState_exit(P0);  // exit action
END_STEP
TRANSITION FROM Wrt_FState TO Init
    := true;
END_TRANSITION

ACTION CkHeadRot_active:


Aux_State_val := ck_state_v( Vision_struct.States_in);
//read register from robot and chek is can read 2 or more correct values 
IF Aux_State_val = VCts.SeparatorRot_R_I THEN
	 I_STATE:= VCts.SeparatorRot_R_I;

//verifies that the vision system has completed its task
ELSIF Aux_State_val = VCts.SeparatorRot_R_F THEN
	
	//read the values processed by the vision system and send to robot
	sep_rot_rigth_data := ck_real_value(Vision_struct.Head_rigth_value);
	//check if all values are correct
	//IF sep_rot_rigth_data.Flag THEN
		//write variables from PLC to CS.UR5 Robot
		//IF wr_real_value(VCts.HEAD_RIGTH_VALUE,sep_rot_rigth_data.Value) THEN
		wr_real_value(VCts.HEAD_RIGTH_VALUE,sep_rot_rigth_data.Value);
		I_STATE := VCts.SeparatorRot_R_F;

		//END_IF
	//END_IF
	
END_IF


//read internal variable and write over output variable
Act_In_State := I_STATE;
END_ACTION

ACTION CkHeadRot_entry:

//start the vision system
wr_state_v(Vcts.SeparatorRot_R);

//write the retain state variable 
Act_Gl_State:=VCts.SeparatorRot_R;
END_ACTION

ACTION CkHeadRot_exit:
//write reset state variables to visiom system.
wr_state_v(RCts.RESET_STATE);
//reset Global state variable
G_STATE := -1;
I_STATE :=-1;

//reset flags vision system to PLC
Vision_struct.States_in.Val1 := -1;
Vision_struct.States_in.Val2 := -1;
Vision_struct.States_in.Val3 := -1;
END_ACTION

ACTION CkHeadRot_L_active:


